Yaskawa INFORM job: DEMO_ROOF_UPPER_0625_3PAINT_53.JBI

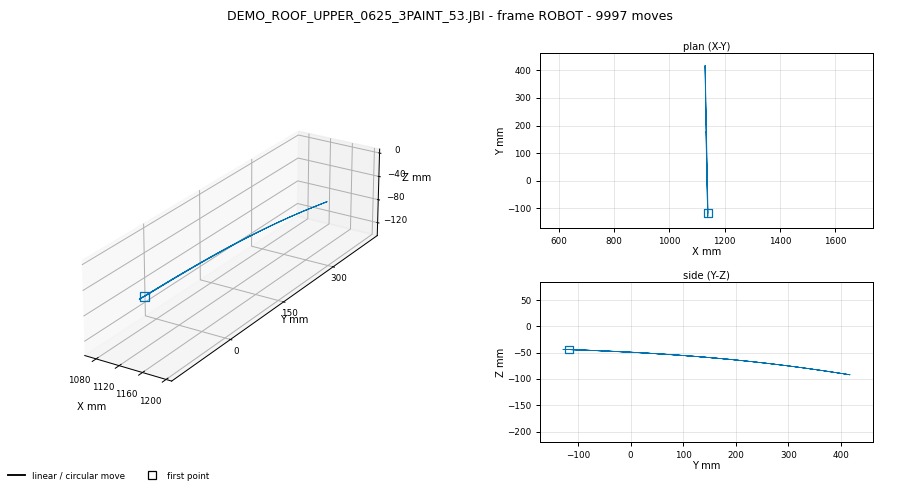
[picture p0: tool path of DEMO_ROOF_UPPER_0625_3PAINT_53.JBI in frame ROBOT, 9997 of 9997 moves have a stored position in this frame; points joined in program order, loops and branches not executed]
/JOB
//NAME DEMO_ROOF_UPPER_0625_3PAINT53
//POS
///NPOS 9997,0,0,0,0,0
///TOOL 0
///USER 0
///POSTYPE ROBOT
///RECTAN
///RCONF 1,0,0,0,0,0,0,0,0,0,0,0,0,0,0,0,0,0,0,0,0,0,0,0
C00000=1140.310,-116.948,-44.068,178.572,6.025,149.504
C00001=1140.305,-116.698,-44.077,178.574,6.025,149.503
C00002=1140.299,-116.448,-44.085,178.576,6.025,149.503
C00003=1140.294,-116.198,-44.094,178.577,6.025,149.502
C00004=1140.288,-115.949,-44.102,178.580,6.026,149.502
C00005=1140.283,-115.699,-44.111,178.581,6.026,149.501
C00006=1140.278,-115.448,-44.119,178.583,6.027,149.501
C00007=1140.272,-115.199,-44.128,178.585,6.027,149.500
C00008=1140.267,-114.949,-44.137,178.587,6.027,149.500
C00009=1140.262,-114.699,-44.146,178.589,6.028,149.499
C00010=1140.256,-114.449,-44.154,178.592,6.028,149.499
C00011=1140.250,-114.200,-44.163,178.594,6.029,149.498
C00012=1140.245,-113.950,-44.171,178.595,6.028,149.498
C00013=1140.240,-113.700,-44.180,178.598,6.029,149.497
C00014=1140.234,-113.450,-44.188,178.599,6.029,149.497
C00015=1140.229,-113.200,-44.197,178.601,6.030,149.496
C00016=1140.224,-112.951,-44.206,178.604,6.031,149.496
C00017=1140.218,-112.701,-44.215,178.605,6.031,149.495
C00018=1140.213,-112.452,-44.223,178.607,6.031,149.495
C00019=1140.208,-112.202,-44.232,178.609,6.031,149.494
C00020=1140.202,-111.951,-44.240,178.611,6.032,149.494
C00021=1140.197,-111.701,-44.249,178.613,6.032,149.493
C00022=1140.191,-111.452,-44.258,178.615,6.033,149.493
C00023=1140.186,-111.202,-44.267,178.617,6.034,149.492
C00024=1140.181,-110.953,-44.276,178.619,6.034,149.492
C00025=1140.176,-110.703,-44.285,178.621,6.034,149.491
C00026=1140.170,-110.452,-44.293,178.623,6.034,149.491
C00027=1140.164,-110.203,-44.301,178.625,6.035,149.490
C00028=1140.159,-109.953,-44.310,178.627,6.035,149.490
C00029=1140.154,-109.703,-44.319,178.629,6.035,149.489
C00030=1140.149,-109.454,-44.328,178.631,6.036,149.489
C00031=1140.143,-109.204,-44.337,178.633,6.036,149.488
C00032=1140.138,-108.955,-44.345,178.635,6.037,149.488
C00033=1140.132,-108.704,-44.355,178.637,6.037,149.487
C00034=1140.127,-108.454,-44.364,178.639,6.037,149.487
C00035=1140.122,-108.205,-44.373,178.641,6.038,149.486
C00036=1140.116,-107.955,-44.381,178.643,6.038,149.486
C00037=1140.111,-107.706,-44.390,178.645,6.039,149.485
C00038=1140.105,-107.455,-44.398,178.647,6.038,149.485
C00039=1140.100,-107.205,-44.407,178.649,6.039,149.484
C00040=1140.095,-106.955,-44.416,178.651,6.040,149.484
C00041=1140.090,-106.706,-44.425,178.653,6.040,149.483
C00042=1140.084,-106.456,-44.434,178.655,6.041,149.483
C00043=1140.078,-106.206,-44.443,178.657,6.041,149.482
C00044=1140.073,-105.956,-44.452,178.659,6.041,149.482
C00045=1140.068,-105.707,-44.461,178.661,6.042,149.481
C00046=1140.063,-105.457,-44.470,178.663,6.042,149.481
C00047=1140.057,-105.207,-44.479,178.665,6.043,149.480
C00048=1140.052,-104.958,-44.487,178.667,6.042,149.479
C00049=1140.047,-104.708,-44.496,178.669,6.043,149.479
C00050=1140.041,-104.458,-44.506,178.671,6.044,149.478
C00051=1140.035,-104.208,-44.514,178.673,6.044,149.478
C00052=1140.030,-103.958,-44.523,178.675,6.045,149.478
C00053=1140.025,-103.709,-44.533,178.677,6.045,149.477
C00054=1140.020,-103.459,-44.542,178.679,6.045,149.477
C00055=1140.014,-103.186,-44.551,178.681,6.046,149.476
C00056=1140.008,-102.915,-44.561,178.684,6.046,149.475
C00057=1140.002,-102.642,-44.571,178.685,6.046,149.475
C00058=1139.996,-102.370,-44.581,178.687,6.047,149.474
C00059=1139.991,-102.120,-44.590,178.690,6.048,149.474
C00060=1139.986,-101.870,-44.599,178.692,6.047,149.473
C00061=1139.981,-101.621,-44.608,178.694,6.048,149.473
C00062=1139.976,-101.371,-44.617,178.696,6.049,149.472
C00063=1139.970,-101.121,-44.627,178.698,6.049,149.472
C00064=1139.964,-100.872,-44.635,178.700,6.050,149.471
C00065=1139.959,-100.622,-44.644,178.702,6.050,149.471
C00066=1139.954,-100.372,-44.653,178.704,6.050,149.470
C00067=1139.948,-100.122,-44.662,178.706,6.051,149.470
C00068=1139.943,-99.872,-44.671,178.709,6.052,149.469
C00069=1139.938,-99.623,-44.681,178.710,6.051,149.469
C00070=1139.933,-99.373,-44.690,178.712,6.052,149.468
C00071=1139.927,-99.123,-44.699,178.714,6.052,149.468
C00072=1139.921,-98.873,-44.708,178.716,6.053,149.467
C00073=1139.916,-98.623,-44.717,178.718,6.054,149.467
C00074=1139.911,-98.374,-44.727,178.720,6.054,149.466
C00075=1139.906,-98.124,-44.736,178.723,6.054,149.465
C00076=1139.900,-97.874,-44.745,178.725,6.055,149.465
C00077=1139.895,-97.625,-44.754,178.726,6.055,149.464
C00078=1139.889,-97.374,-44.763,178.729,6.055,149.464
C00079=1139.884,-97.125,-44.773,178.731,6.056,149.463
C00080=1139.879,-96.875,-44.782,178.732,6.056,149.463
C00081=1139.873,-96.625,-44.791,178.735,6.057,149.463
C00082=1139.868,-96.375,-44.800,178.737,6.057,149.462
C00083=1139.862,-96.126,-44.809,178.739,6.057,149.461
C00084=1139.857,-95.876,-44.819,178.741,6.058,149.461
C00085=1139.852,-95.626,-44.828,178.743,6.058,149.460
C00086=1139.847,-95.376,-44.837,178.745,6.059,149.460
C00087=1139.841,-95.127,-44.847,178.747,6.060,149.459
C00088=1139.836,-94.877,-44.856,178.749,6.059,149.459
C00089=1139.831,-94.627,-44.865,178.751,6.060,149.458
C00090=1139.825,-94.377,-44.874,178.754,6.061,149.458
C00091=1139.820,-94.128,-44.884,178.755,6.061,149.457
C00092=1139.815,-93.878,-44.893,178.757,6.061,149.457
C00093=1139.809,-93.628,-44.902,178.760,6.062,149.456
C00094=1139.804,-93.378,-44.912,178.761,6.062,149.456
C00095=1139.799,-93.129,-44.921,178.763,6.063,149.455
C00096=1139.793,-92.878,-44.930,178.766,6.063,149.455
C00097=1139.788,-92.629,-44.940,178.768,6.063,149.454
C00098=1139.782,-92.379,-44.950,178.770,6.064,149.454
C00099=1139.777,-92.129,-44.959,178.772,6.065,149.453
C00100=1139.772,-91.880,-44.968,178.774,6.065,149.453
C00101=1139.766,-91.630,-44.978,178.776,6.065,149.452
C00102=1139.761,-91.380,-44.987,178.778,6.066,149.451
C00103=1139.755,-91.130,-44.997,178.780,6.066,149.451
C00104=1139.750,-90.880,-45.006,178.782,6.066,149.450
C00105=1139.745,-90.631,-45.015,178.784,6.067,149.450
C00106=1139.739,-90.381,-45.025,178.787,6.068,149.449
C00107=1139.734,-90.131,-45.034,178.788,6.068,149.449
C00108=1139.729,-89.882,-45.044,178.791,6.068,149.448
C00109=1139.724,-89.632,-45.053,178.793,6.069,149.448
C00110=1139.718,-89.382,-45.063,178.795,6.069,149.447
C00111=1139.713,-89.132,-45.072,178.797,6.070,149.447
C00112=1139.707,-88.883,-45.082,178.799,6.071,149.446
C00113=1139.702,-88.633,-45.091,178.801,6.070,149.446
C00114=1139.697,-88.382,-45.101,178.803,6.071,149.445
C00115=1139.692,-88.133,-45.110,178.806,6.072,149.445
C00116=1139.687,-87.883,-45.119,178.807,6.072,149.444
C00117=1139.681,-87.634,-45.130,178.809,6.072,149.444
C00118=1139.676,-87.384,-45.138,178.812,6.073,149.443
C00119=1139.670,-87.134,-45.149,178.814,6.073,149.443
C00120=1139.665,-86.884,-45.158,178.816,6.073,149.442
C00121=1139.660,-86.635,-45.168,178.818,6.074,149.442
C00122=1139.654,-86.385,-45.177,178.820,6.075,149.441
C00123=1139.649,-86.135,-45.187,178.822,6.075,149.441
C00124=1139.644,-85.886,-45.196,178.824,6.075,149.440
C00125=1139.639,-85.635,-45.206,178.827,6.076,149.439
C00126=1139.633,-85.385,-45.215,178.828,6.076,149.439
C00127=1139.628,-85.136,-45.225,178.830,6.077,149.438
C00128=1139.622,-84.886,-45.236,178.833,6.078,149.438
C00129=1139.617,-84.636,-45.245,178.835,6.078,149.437
C00130=1139.611,-84.387,-45.255,178.837,6.078,149.437
C00131=1139.606,-84.137,-45.264,178.839,6.079,149.436
C00132=1139.601,-83.888,-45.274,178.841,6.079,149.436
C00133=1139.596,-83.638,-45.283,178.843,6.079,149.435
C00134=1139.591,-83.387,-45.293,178.845,6.080,149.435
C00135=1139.586,-83.138,-45.303,178.848,6.080,149.434
C00136=1139.580,-82.888,-45.312,178.850,6.081,149.434
C00137=1139.574,-82.639,-45.323,178.851,6.081,149.433
C00138=1139.569,-82.389,-45.332,178.854,6.082,149.433
C00139=1139.563,-82.139,-45.342,178.856,6.082,149.432
C00140=1139.559,-81.890,-45.351,178.858,6.082,149.431
C00141=1139.553,-81.639,-45.361,178.860,6.083,149.431
C00142=1139.548,-81.389,-45.371,178.862,6.084,149.430
C00143=1139.543,-81.140,-45.381,178.865,6.085,149.430
C00144=1139.537,-80.890,-45.391,178.867,6.084,149.429
C00145=1139.532,-80.641,-45.400,178.869,6.085,149.429
C00146=1139.526,-80.391,-45.410,178.871,6.086,149.428
C00147=1139.521,-80.140,-45.420,178.873,6.086,149.428
C00148=1139.516,-79.891,-45.430,178.875,6.086,149.427
C00149=1139.511,-79.642,-45.440,178.877,6.087,149.427
C00150=1139.505,-79.392,-45.450,178.880,6.088,149.426
C00151=1139.500,-79.142,-45.459,178.882,6.088,149.426
C00152=1139.495,-78.892,-45.470,178.883,6.088,149.425
C00153=1139.489,-78.642,-45.480,178.886,6.089,149.425
C00154=1139.484,-78.393,-45.489,178.888,6.089,149.424
C00155=1139.479,-78.143,-45.499,178.891,6.090,149.424
C00156=1139.473,-77.894,-45.509,178.892,6.090,149.423
C00157=1139.468,-77.644,-45.518,178.894,6.091,149.423
C00158=1139.463,-77.393,-45.529,178.897,6.091,149.422
C00159=1139.456,-77.123,-45.540,178.899,6.092,149.421
C00160=1139.451,-76.851,-45.550,178.901,6.093,149.421
C00161=1139.446,-76.579,-45.561,178.904,6.093,149.420
C00162=1139.440,-76.308,-45.573,178.906,6.093,149.420
C00163=1139.434,-76.058,-45.583,178.908,6.094,149.419
C00164=1139.429,-75.808,-45.592,178.910,6.094,149.419
C00165=1139.423,-75.559,-45.602,178.913,6.095,149.418
C00166=1139.418,-75.309,-45.612,178.914,6.095,149.418
C00167=1139.413,-75.059,-45.622,178.916,6.096,149.417
C00168=1139.408,-74.810,-45.632,178.919,6.096,149.416
C00169=1139.402,-74.560,-45.642,178.921,6.097,149.416
C00170=1139.396,-74.310,-45.652,178.924,6.098,149.415
C00171=1139.391,-74.060,-45.663,178.925,6.098,149.415
C00172=1139.386,-73.811,-45.672,178.928,6.098,149.414
C00173=1139.381,-73.561,-45.682,178.930,6.099,149.414
C00174=1139.375,-73.312,-45.693,178.932,6.100,149.413
C00175=1139.370,-73.061,-45.703,178.934,6.100,149.413
C00176=1139.365,-72.812,-45.713,178.936,6.100,149.412
C00177=1139.360,-72.562,-45.722,178.939,6.101,149.412
C00178=1139.355,-72.312,-45.733,178.941,6.101,149.411
C00179=1139.349,-72.062,-45.743,178.942,6.101,149.411
C00180=1139.343,-71.813,-45.753,178.945,6.102,149.410
C00181=1139.338,-71.563,-45.763,178.947,6.103,149.409
C00182=1139.333,-71.313,-45.773,178.949,6.103,149.409
C00183=1139.328,-71.064,-45.784,178.952,6.104,149.408
C00184=1139.322,-70.814,-45.794,178.953,6.104,149.408
C00185=1139.317,-70.564,-45.804,178.956,6.104,149.407
C00186=1139.312,-70.314,-45.815,178.958,6.105,149.407
C00187=1139.307,-70.065,-45.824,178.960,6.106,149.406
C00188=1139.302,-69.815,-45.835,178.963,6.107,149.406
C00189=1139.296,-69.565,-45.845,178.965,6.106,149.405
C00190=1139.291,-69.316,-45.855,178.967,6.107,149.405
C00191=1139.285,-69.066,-45.865,178.969,6.108,149.404
C00192=1139.280,-68.816,-45.876,178.971,6.109,149.404
C00193=1139.274,-68.566,-45.886,178.974,6.109,149.403
C00194=1139.269,-68.317,-45.896,178.975,6.109,149.402
C00195=1139.265,-68.067,-45.906,178.978,6.110,149.402
C00196=1139.259,-67.817,-45.917,178.980,6.110,149.401
C00197=1139.254,-67.567,-45.927,178.982,6.111,149.401
C00198=1139.248,-67.317,-45.937,178.985,6.112,149.400
C00199=1139.243,-67.068,-45.948,178.986,6.112,149.400
C00200=1139.238,-66.818,-45.958,178.989,6.112,149.399
C00201=1139.232,-66.568,-45.968,178.991,6.113,149.399
C00202=1139.227,-66.319,-45.979,178.993,6.114,149.398
C00203=1139.222,-66.068,-45.989,178.996,6.114,149.398
C00204=1139.216,-65.819,-45.999,178.998,6.114,149.397
C00205=1139.211,-65.570,-46.009,179.000,6.115,149.396
C00206=1139.206,-65.319,-46.020,179.002,6.115,149.396
C00207=1139.201,-65.070,-46.031,179.004,6.116,149.396
C00208=1139.196,-64.820,-46.041,179.007,6.117,149.395
C00209=1139.190,-64.571,-46.051,179.008,6.117,149.394
C00210=1139.185,-64.321,-46.062,179.011,6.117,149.394
C00211=1139.180,-64.071,-46.072,179.013,6.118,149.393
C00212=1139.174,-63.821,-46.082,179.015,6.118,149.393
C00213=1139.169,-63.571,-46.093,179.018,6.119,149.392
C00214=1139.164,-63.322,-46.104,179.020,6.120,149.392
C00215=1139.158,-63.073,-46.114,179.021,6.120,149.391
C00216=1139.153,-62.822,-46.125,179.024,6.120,149.391
C00217=1139.148,-62.573,-46.135,179.026,6.121,149.390
C00218=1139.143,-62.323,-46.145,179.028,6.122,149.390
C00219=1139.137,-62.073,-46.156,179.031,6.122,149.389
C00220=1139.132,-61.823,-46.167,179.033,6.123,149.388
C00221=1139.127,-61.574,-46.177,179.035,6.123,149.388
C00222=1139.121,-61.324,-46.187,179.037,6.124,149.387
C00223=1139.116,-61.074,-46.198,179.040,6.124,149.387
C00224=1139.111,-60.825,-46.209,179.042,6.125,149.386
C00225=1139.106,-60.575,-46.219,179.044,6.126,149.386
C00226=1139.100,-60.325,-46.230,179.047,6.126,149.385
C00227=1139.095,-60.075,-46.240,179.048,6.126,149.385
C00228=1139.090,-59.826,-46.251,179.051,6.127,149.384
C00229=1139.085,-59.576,-46.262,179.053,6.128,149.384
C00230=1139.079,-59.326,-46.272,179.055,6.128,149.383
C00231=1139.074,-59.076,-46.282,179.058,6.129,149.382
C00232=1139.068,-58.827,-46.294,179.060,6.130,149.382
C00233=1139.063,-58.577,-46.305,179.062,6.130,149.381
C00234=1139.058,-58.327,-46.315,179.064,6.130,149.381
C00235=1139.053,-58.077,-46.326,179.066,6.131,149.380
C00236=1139.047,-57.828,-46.336,179.069,6.131,149.380
C00237=1139.042,-57.578,-46.347,179.071,6.132,149.379
C00238=1139.037,-57.329,-46.358,179.073,6.133,149.379
C00239=1139.032,-57.079,-46.368,179.076,6.133,149.378
C00240=1139.026,-56.829,-46.379,179.078,6.134,149.377
C00241=1139.022,-56.579,-46.390,179.080,6.134,149.377
C00242=1139.016,-56.330,-46.400,179.082,6.135,149.376
C00243=1139.011,-56.080,-46.412,179.084,6.135,149.376
C00244=1139.005,-55.830,-46.422,179.087,6.136,149.375
C00245=1139.000,-55.580,-46.433,179.089,6.136,149.375
C00246=1138.995,-55.331,-46.444,179.091,6.137,149.374
C00247=1138.990,-55.081,-46.454,179.094,6.138,149.374
C00248=1138.985,-54.832,-46.465,179.096,6.138,149.373
C00249=1138.980,-54.582,-46.476,179.098,6.138,149.373
C00250=1138.973,-54.332,-46.486,179.100,6.139,149.372
C00251=1138.969,-54.082,-46.498,179.103,6.140,149.371
C00252=1138.964,-53.832,-46.508,179.105,6.140,149.371
C00253=1138.958,-53.583,-46.519,179.107,6.141,149.371
C00254=1138.953,-53.333,-46.530,179.110,6.141,149.370
C00255=1138.947,-53.084,-46.541,179.112,6.142,149.369
C00256=1138.942,-52.833,-46.552,179.114,6.143,149.369
C00257=1138.937,-52.584,-46.563,179.116,6.143,149.368
C00258=1138.932,-52.334,-46.573,179.118,6.143,149.368
C00259=1138.927,-52.085,-46.584,179.120,6.144,149.367
C00260=1138.921,-51.835,-46.596,179.123,6.145,149.367
C00261=1138.916,-51.585,-46.607,179.125,6.145,149.366
C00262=1138.911,-51.336,-46.617,179.127,6.146,149.366
C00263=1138.905,-51.065,-46.629,179.130,6.146,149.365
C00264=1138.899,-50.794,-46.641,179.132,6.147,149.364
C00265=1138.894,-50.524,-46.653,179.135,6.148,149.364
C00266=1138.888,-50.253,-46.665,179.137,6.148,149.363
C00267=1138.883,-50.003,-46.675,179.139,6.149,149.363
C00268=1138.877,-49.753,-46.687,179.142,6.150,149.362
C00269=1138.872,-49.503,-46.698,179.144,6.150,149.362
C00270=1138.867,-49.254,-46.709,179.146,6.151,149.361
C00271=1138.861,-49.003,-46.720,179.149,6.151,149.360
C00272=1138.856,-48.755,-46.731,179.151,6.152,149.360
C00273=1138.851,-48.505,-46.742,179.153,6.152,149.359
C00274=1138.846,-48.255,-46.753,179.155,6.153,149.359
C00275=1138.840,-48.005,-46.764,179.158,6.153,149.358
C00276=1138.836,-47.756,-46.775,179.160,6.154,149.358
C00277=1138.831,-47.506,-46.786,179.162,6.155,149.357
C00278=1138.825,-47.256,-46.798,179.165,6.155,149.357
C00279=1138.820,-47.006,-46.808,179.167,6.156,149.356
C00280=1138.814,-46.757,-46.819,179.169,6.157,149.356
C00281=1138.809,-46.507,-46.831,179.172,6.157,149.355
C00282=1138.804,-46.257,-46.841,179.174,6.158,149.354
C00283=1138.799,-46.008,-46.852,179.176,6.159,149.354
C00284=1138.793,-45.758,-46.864,179.179,6.159,149.353
C00285=1138.788,-45.508,-46.876,179.181,6.160,149.353
C00286=1138.782,-45.259,-46.886,179.183,6.160,149.352
C00287=1138.777,-45.009,-46.898,179.185,6.160,149.352
C00288=1138.773,-44.759,-46.909,179.188,6.161,149.351
C00289=1138.767,-44.509,-46.920,179.190,6.162,149.351
C00290=1138.762,-44.260,-46.931,179.192,6.162,149.350
C00291=1138.757,-44.010,-46.942,179.195,6.163,149.349
C00292=1138.752,-43.760,-46.954,179.197,6.164,149.349
C00293=1138.746,-43.511,-46.964,179.199,6.164,149.348
C00294=1138.740,-43.261,-46.976,179.202,6.165,149.348
C00295=1138.736,-43.011,-46.988,179.204,6.166,149.347
C00296=1138.731,-42.762,-46.999,179.206,6.167,149.347
C00297=1138.725,-42.512,-47.010,179.209,6.167,149.346
C00298=1138.720,-42.262,-47.021,179.211,6.168,149.346
C00299=1138.715,-42.012,-47.033,179.213,6.169,149.345
C00300=1138.709,-41.763,-47.044,179.216,6.169,149.344
C00301=1138.704,-41.513,-47.056,179.218,6.170,149.344
C00302=1138.699,-41.264,-47.067,179.220,6.171,149.344
C00303=1138.694,-41.013,-47.078,179.223,6.171,149.343
C00304=1138.688,-40.764,-47.089,179.224,6.171,149.342
C00305=1138.683,-40.514,-47.101,179.226,6.172,149.342
C00306=1138.678,-40.265,-47.112,179.229,6.172,149.341
C00307=1138.672,-40.015,-47.124,179.231,6.173,149.341
C00308=1138.667,-39.766,-47.135,179.234,6.174,149.340
C00309=1138.662,-39.516,-47.147,179.236,6.174,149.340
C00310=1138.657,-39.266,-47.158,179.238,6.175,149.339
C00311=1138.651,-39.016,-47.169,179.241,6.176,149.339
C00312=1138.646,-38.767,-47.180,179.243,6.176,149.338
C00313=1138.641,-38.517,-47.192,179.245,6.177,149.337
C00314=1138.636,-38.267,-47.204,179.248,6.178,149.337
C00315=1138.631,-38.017,-47.215,179.250,6.178,149.336
C00316=1138.625,-37.768,-47.226,179.252,6.179,149.336
C00317=1138.620,-37.518,-47.238,179.255,6.180,149.335
C00318=1138.615,-37.269,-47.249,179.257,6.180,149.335
C00319=1138.610,-37.019,-47.261,179.260,6.181,149.334
C00320=1138.605,-36.769,-47.273,179.262,6.182,149.334
C00321=1138.599,-36.520,-47.284,179.264,6.182,149.333
C00322=1138.594,-36.270,-47.296,179.267,6.183,149.332
C00323=1138.589,-36.020,-47.307,179.269,6.183,149.332
C00324=1138.584,-35.770,-47.319,179.271,6.184,149.331
C00325=1138.579,-35.521,-47.331,179.274,6.185,149.331
C00326=1138.573,-35.272,-47.342,179.276,6.185,149.330
C00327=1138.567,-35.022,-47.354,179.278,6.186,149.330
C00328=1138.563,-34.772,-47.365,179.281,6.187,149.329
C00329=1138.557,-34.522,-47.377,179.283,6.187,149.329
C00330=1138.553,-34.272,-47.388,179.285,6.188,149.328
C00331=1138.547,-34.023,-47.400,179.288,6.189,149.327
C00332=1138.541,-33.773,-47.412,179.290,6.189,149.327
C00333=1138.536,-33.524,-47.423,179.293,6.190,149.326
C00334=1138.531,-33.274,-47.435,179.295,6.191,149.326
C00335=1138.526,-33.024,-47.447,179.297,6.191,149.325
C00336=1138.521,-32.774,-47.458,179.300,6.192,149.325
C00337=1138.515,-32.524,-47.470,179.302,6.193,149.324
C00338=1138.511,-32.275,-47.481,179.304,6.193,149.324
C00339=1138.505,-32.026,-47.494,179.307,6.194,149.323
C00340=1138.500,-31.776,-47.505,179.309,6.195,149.323
C00341=1138.495,-31.526,-47.517,179.311,6.195,149.322
C00342=1138.489,-31.277,-47.529,179.314,6.196,149.321
C00343=1138.484,-31.027,-47.541,179.316,6.196,149.321
C00344=1138.479,-30.777,-47.552,179.318,6.197,149.320
C00345=1138.474,-30.527,-47.564,179.321,6.198,149.320
C00346=1138.469,-30.278,-47.576,179.323,6.198,149.319
C00347=1138.463,-30.028,-47.588,179.325,6.199,149.319
C00348=1138.458,-29.779,-47.599,179.328,6.200,149.318
C00349=1138.453,-29.529,-47.611,179.330,6.200,149.318
C00350=1138.447,-29.279,-47.623,179.333,6.201,149.317
C00351=1138.442,-29.030,-47.635,179.335,6.202,149.316
C00352=1138.437,-28.780,-47.647,179.337,6.202,149.316
C00353=1138.432,-28.530,-47.659,179.340,6.203,149.315
C00354=1138.427,-28.280,-47.671,179.342,6.204,149.315
C00355=1138.422,-28.031,-47.683,179.344,6.204,149.314
C00356=1138.417,-27.781,-47.694,179.347,6.205,149.314
C00357=1138.411,-27.531,-47.706,179.349,6.206,149.313
C00358=1138.406,-27.281,-47.718,179.351,6.206,149.313
C00359=1138.401,-27.032,-47.731,179.354,6.207,149.312
C00360=1138.396,-26.782,-47.742,179.356,6.208,149.311
C00361=1138.391,-26.532,-47.754,179.359,6.209,149.311
C00362=1138.386,-26.283,-47.767,179.361,6.210,149.310
C00363=1138.380,-26.033,-47.778,179.363,6.210,149.310
C00364=1138.375,-25.784,-47.790,179.366,6.211,149.309
C00365=1138.370,-25.534,-47.802,179.368,6.212,149.309
C00366=1138.365,-25.284,-47.814,179.370,6.212,149.308
C00367=1138.359,-25.015,-47.827,179.373,6.213,149.307
C00368=1138.354,-24.744,-47.840,179.375,6.214,149.307
C00369=1138.347,-24.474,-47.853,179.378,6.214,149.306
C00370=1138.342,-24.204,-47.866,179.381,6.216,149.306
C00371=1138.337,-23.955,-47.879,179.383,6.216,149.305
C00372=1138.331,-23.705,-47.890,179.386,6.217,149.305
C00373=1138.326,-23.455,-47.902,179.388,6.217,149.304
C00374=1138.321,-23.206,-47.914,179.390,6.218,149.304
C00375=1138.316,-22.956,-47.926,179.393,6.219,149.303
C00376=1138.311,-22.707,-47.939,179.395,6.219,149.303
C00377=1138.305,-22.457,-47.951,179.397,6.220,149.302
C00378=1138.300,-22.207,-47.963,179.400,6.221,149.301
C00379=1138.295,-21.957,-47.975,179.402,6.221,149.301
C00380=1138.289,-21.707,-47.987,179.405,6.222,149.300
C00381=1138.284,-21.458,-48.000,179.407,6.223,149.300
C00382=1138.280,-21.208,-48.011,179.409,6.223,149.299
C00383=1138.274,-20.959,-48.024,179.412,6.225,149.299
C00384=1138.269,-20.709,-48.035,179.414,6.225,149.298
C00385=1138.264,-20.460,-48.048,179.417,6.226,149.297
C00386=1138.258,-20.210,-48.060,179.419,6.227,149.297
C00387=1138.253,-19.961,-48.073,179.421,6.227,149.296
C00388=1138.248,-19.710,-48.085,179.424,6.228,149.296
C00389=1138.243,-19.461,-48.097,179.426,6.229,149.295
C00390=1138.238,-19.211,-48.109,179.428,6.229,149.295
C00391=1138.233,-18.961,-48.122,179.431,6.230,149.294
C00392=1138.228,-18.712,-48.134,179.433,6.231,149.294
C00393=1138.222,-18.462,-48.146,179.436,6.231,149.293
C00394=1138.217,-18.213,-48.159,179.439,6.233,149.293
C00395=1138.212,-17.963,-48.171,179.441,6.233,149.292
C00396=1138.207,-17.714,-48.183,179.444,6.234,149.291
C00397=1138.201,-17.464,-48.195,179.446,6.235,149.291
C00398=1138.196,-17.214,-48.208,179.448,6.235,149.290
C00399=1138.191,-16.965,-48.221,179.451,6.236,149.290
C00400=1138.186,-16.714,-48.233,179.453,6.237,149.289
C00401=1138.181,-16.465,-48.245,179.455,6.237,149.289
C00402=1138.175,-16.215,-48.257,179.458,6.238,149.288
C00403=1138.170,-15.966,-48.270,179.460,6.239,149.288
C00404=1138.165,-15.717,-48.282,179.463,6.240,149.287
C00405=1138.160,-15.467,-48.294,179.465,6.241,149.286
C00406=1138.155,-15.217,-48.307,179.467,6.241,149.286
C00407=1138.150,-14.967,-48.320,179.470,6.242,149.285
C00408=1138.145,-14.717,-48.332,179.472,6.243,149.285
C00409=1138.140,-14.468,-48.344,179.474,6.243,149.284
C00410=1138.134,-14.219,-48.357,179.477,6.244,149.284
C00411=1138.129,-13.969,-48.370,179.479,6.245,149.283
C00412=1138.123,-13.719,-48.382,179.481,6.245,149.283
C00413=1138.118,-13.470,-48.395,179.485,6.247,149.282
C00414=1138.114,-13.220,-48.408,179.487,6.247,149.282
C00415=1138.108,-12.970,-48.420,179.490,6.248,149.281
C00416=1138.103,-12.721,-48.432,179.492,6.249,149.280
C00417=1138.098,-12.471,-48.445,179.494,6.249,149.280
C00418=1138.093,-12.222,-48.457,179.497,6.250,149.279
C00419=1138.088,-11.972,-48.470,179.499,6.251,149.279
C00420=1138.082,-11.722,-48.483,179.501,6.252,149.278
C00421=1138.077,-11.472,-48.495,179.504,6.253,149.278
C00422=1138.072,-11.223,-48.508,179.506,6.253,149.277
C00423=1138.067,-10.974,-48.521,179.509,6.254,149.277
C00424=1138.062,-10.724,-48.534,179.511,6.255,149.276
C00425=1138.057,-10.474,-48.545,179.513,6.255,149.275
C00426=1138.052,-10.224,-48.558,179.516,6.256,149.275
C00427=1138.046,-9.975,-48.571,179.519,6.257,149.274
C00428=1138.041,-9.725,-48.584,179.521,6.258,149.274
C00429=1138.036,-9.475,-48.597,179.524,6.259,149.273
C00430=1138.031,-9.226,-48.609,179.526,6.260,149.273
C00431=1138.026,-8.976,-48.621,179.528,6.260,149.272
C00432=1138.020,-8.727,-48.634,179.531,6.261,149.272
C00433=1138.015,-8.477,-48.647,179.533,6.262,149.271
C00434=1138.010,-8.227,-48.660,179.536,6.263,149.271
C00435=1138.005,-7.978,-48.673,179.538,6.264,149.270
C00436=1138.000,-7.729,-48.685,179.540,6.264,149.269
C00437=1137.995,-7.478,-48.699,179.543,6.265,149.269
C00438=1137.989,-7.229,-48.711,179.545,6.266,149.268
C00439=1137.984,-6.980,-48.724,179.547,6.266,149.268
C00440=1137.979,-6.730,-48.737,179.551,6.268,149.267
C00441=1137.974,-6.480,-48.750,179.553,6.268,149.267
C00442=1137.969,-6.231,-48.763,179.555,6.269,149.266
C00443=1137.964,-5.981,-48.775,179.558,6.270,149.266
C00444=1137.959,-5.731,-48.788,179.560,6.270,149.265
C00445=1137.953,-5.482,-48.802,179.563,6.272,149.265
C00446=1137.948,-5.232,-48.814,179.565,6.272,149.264
C00447=1137.943,-4.983,-48.827,179.568,6.273,149.263
C00448=1137.938,-4.733,-48.840,179.570,6.274,149.263
C00449=1137.933,-4.483,-48.853,179.572,6.274,149.262
C00450=1137.928,-4.234,-48.866,179.575,6.275,149.262
C00451=1137.922,-3.984,-48.879,179.578,6.276,149.261
C00452=1137.917,-3.734,-48.892,179.580,6.277,149.261
C00453=1137.912,-3.485,-48.904,179.582,6.278,149.260
C00454=1137.907,-3.235,-48.918,179.585,6.278,149.259
C00455=1137.902,-2.985,-48.930,179.587,6.279,149.259
C00456=1137.896,-2.736,-48.943,179.590,6.280,149.258
C00457=1137.891,-2.486,-48.957,179.592,6.281,149.258
C00458=1137.886,-2.236,-48.969,179.595,6.282,149.257
C00459=1137.881,-1.987,-48.982,179.597,6.283,149.257
C00460=1137.876,-1.737,-48.996,179.599,6.283,149.256
C00461=1137.871,-1.488,-49.009,179.602,6.285,149.256
C00462=1137.865,-1.239,-49.022,179.605,6.285,149.255
C00463=1137.861,-0.989,-49.035,179.607,6.286,149.255
C00464=1137.855,-0.739,-49.047,179.609,6.287,149.254
C00465=1137.850,-0.489,-49.061,179.612,6.287,149.253
C00466=1137.845,-0.240,-49.074,179.615,6.289,149.253
C00467=1137.839,0.009,-49.088,179.617,6.289,149.252
C00468=1137.835,0.259,-49.100,179.619,6.290,149.252
C00469=1137.829,0.509,-49.114,179.622,6.291,149.251
C00470=1137.824,0.758,-49.126,179.624,6.291,149.251
C00471=1137.819,1.028,-49.141,179.627,6.293,149.250
C00472=1137.814,1.298,-49.155,179.630,6.293,149.250
C00473=1137.808,1.568,-49.169,179.633,6.295,149.249
C00474=1137.802,1.836,-49.184,179.635,6.295,149.248
C00475=1137.797,2.086,-49.197,179.637,6.296,149.248
C00476=1137.791,2.336,-49.210,179.641,6.297,149.247
C00477=1137.787,2.585,-49.224,179.643,6.298,149.247
C00478=1137.781,2.835,-49.237,179.645,6.299,149.246
C00479=1137.776,3.084,-49.249,179.648,6.300,149.246
C00480=1137.772,3.334,-49.262,179.650,6.300,149.245
C00481=1137.766,3.583,-49.276,179.653,6.302,149.245
C00482=1137.761,3.834,-49.290,179.655,6.302,149.244
C00483=1137.756,4.083,-49.303,179.657,6.303,149.244
C00484=1137.751,4.333,-49.317,179.660,6.304,149.243
C00485=1137.746,4.582,-49.329,179.663,6.305,149.242
C00486=1137.740,4.832,-49.343,179.665,6.306,149.242
C00487=1137.736,5.081,-49.356,179.668,6.306,149.241
C00488=1137.730,5.331,-49.370,179.670,6.307,149.241
C00489=1137.725,5.580,-49.383,179.673,6.309,149.240
C00490=1137.720,5.830,-49.396,179.675,6.309,149.240
C00491=1137.715,6.080,-49.409,179.677,6.310,149.239
C00492=1137.710,6.329,-49.423,179.680,6.311,149.239
C00493=1137.704,6.579,-49.437,179.683,6.312,149.238
C00494=1137.699,6.828,-49.450,179.685,6.313,149.238
C00495=1137.694,7.078,-49.464,179.688,6.313,149.237
C00496=1137.689,7.327,-49.476,179.690,6.314,149.236
C00497=1137.684,7.577,-49.491,179.693,6.316,149.236
C00498=1137.678,7.827,-49.504,179.695,6.316,149.235
C00499=1137.674,8.076,-49.517,179.697,6.317,149.235
C00500=1137.668,8.326,-49.531,179.700,6.319,149.234
C00501=1137.664,8.575,-49.544,179.703,6.319,149.234
C00502=1137.659,8.826,-49.558,179.705,6.320,149.233
C00503=1137.653,9.075,-49.572,179.708,6.320,149.232
C00504=1137.649,9.325,-49.585,179.711,6.322,149.232
C00505=1137.643,9.574,-49.599,179.713,6.323,149.232
C00506=1137.638,9.824,-49.612,179.715,6.323,149.231
C00507=1137.633,10.073,-49.626,179.718,6.324,149.230
C00508=1137.628,10.323,-49.639,179.720,6.326,149.230
C00509=1137.622,10.572,-49.653,179.723,6.326,149.229
C00510=1137.618,10.821,-49.667,179.725,6.327,149.229
C00511=1137.612,11.071,-49.680,179.728,6.328,149.228
C00512=1137.607,11.321,-49.694,179.731,6.329,149.228
C00513=1137.603,11.571,-49.707,179.733,6.330,149.227
C00514=1137.597,11.820,-49.721,179.735,6.330,149.226
C00515=1137.592,12.070,-49.735,179.738,6.332,149.226
C00516=1137.586,12.319,-49.749,179.740,6.332,149.226
C00517=1137.582,12.568,-49.762,179.743,6.333,149.225
C00518=1137.577,12.819,-49.776,179.746,6.335,149.224
C00519=1137.571,13.068,-49.790,179.748,6.335,149.224
C00520=1137.566,13.317,-49.804,179.751,6.336,149.223
C00521=1137.561,13.567,-49.817,179.753,6.337,149.223
C00522=1137.556,13.816,-49.831,179.756,6.338,149.222
C00523=1137.551,14.066,-49.845,179.758,6.339,149.222
C00524=1137.545,14.316,-49.858,179.760,6.339,149.221
C00525=1137.541,14.565,-49.872,179.764,6.341,149.221
C00526=1137.536,14.814,-49.886,179.766,6.341,149.220
C00527=1137.530,15.065,-49.899,179.768,6.342,149.220
C00528=1137.525,15.314,-49.914,179.771,6.344,149.219
C00529=1137.520,15.563,-49.928,179.773,6.344,149.218
C00530=1137.516,15.813,-49.941,179.776,6.345,149.218
C00531=1137.510,16.063,-49.955,179.779,6.346,149.217
C00532=1137.505,16.312,-49.969,179.781,6.347,149.217
C00533=1137.500,16.562,-49.983,179.783,6.348,149.216
C00534=1137.495,16.811,-49.997,179.786,6.349,149.216
C00535=1137.489,17.060,-50.011,179.789,6.350,149.215
C00536=1137.485,17.310,-50.024,179.791,6.351,149.215
C00537=1137.480,17.560,-50.039,179.794,6.352,149.214
C00538=1137.474,17.809,-50.052,179.796,6.353,149.214
C00539=1137.469,18.059,-50.067,179.799,6.353,149.213
C00540=1137.464,18.309,-50.081,179.802,6.355,149.213
C00541=1137.458,18.558,-50.094,179.804,6.356,149.212
C00542=1137.454,18.808,-50.108,179.806,6.356,149.211
C00543=1137.449,19.058,-50.123,179.809,6.358,149.211
C00544=1137.444,19.306,-50.136,179.811,6.359,149.210
C00545=1137.439,19.556,-50.150,179.814,6.359,149.210
C00546=1137.434,19.806,-50.165,179.817,6.361,149.209
C00547=1137.429,20.056,-50.179,179.819,6.362,149.209
C00548=1137.423,20.305,-50.193,179.822,6.362,149.208
C00549=1137.418,20.555,-50.206,179.824,6.364,149.208
C00550=1137.413,20.805,-50.221,179.827,6.364,149.207
C00551=1137.408,21.054,-50.235,179.829,6.365,149.207
C00552=1137.403,21.303,-50.249,179.832,6.366,149.206
C00553=1137.398,21.553,-50.263,179.835,6.367,149.205
C00554=1137.393,21.803,-50.277,179.837,6.369,149.205
C00555=1137.388,22.052,-50.292,179.840,6.369,149.205
C00556=1137.382,22.301,-50.306,179.842,6.370,149.204
C00557=1137.377,22.551,-50.320,179.845,6.371,149.203
C00558=1137.372,22.801,-50.334,179.847,6.372,149.203
C00559=1137.367,23.051,-50.348,179.850,6.373,149.202
C00560=1137.362,23.300,-50.362,179.853,6.374,149.202
C00561=1137.357,23.549,-50.377,179.855,6.375,149.201
C00562=1137.352,23.799,-50.391,179.858,6.376,149.201
C00563=1137.347,24.049,-50.405,179.860,6.377,149.200
C00564=1137.341,24.298,-50.419,179.862,6.378,149.200
C00565=1137.336,24.547,-50.433,179.866,6.379,149.199
C00566=1137.331,24.797,-50.448,179.868,6.380,149.199
C00567=1137.327,25.046,-50.463,179.870,6.380,149.198
C00568=1137.322,25.296,-50.477,179.873,6.382,149.197
C00569=1137.316,25.545,-50.491,179.875,6.383,149.197
C00570=1137.311,25.795,-50.505,179.879,6.384,149.196
C00571=1137.306,26.044,-50.519,179.881,6.385,149.196
C00572=1137.301,26.294,-50.534,179.883,6.386,149.195
C00573=1137.296,26.544,-50.548,179.886,6.387,149.195
C00574=1137.292,26.793,-50.562,179.888,6.388,149.194
C00575=1137.285,27.062,-50.578,179.892,6.389,149.194
C00576=1137.280,27.331,-50.594,179.894,6.390,149.193
C00577=1137.274,27.600,-50.609,179.897,6.391,149.192
C00578=1137.269,27.869,-50.625,179.900,6.393,149.192
C00579=1137.264,28.119,-50.639,179.902,6.394,149.192
C00580=1137.259,28.369,-50.654,179.905,6.394,149.191
C00581=1137.254,28.618,-50.668,179.907,6.396,149.190
C00582=1137.249,28.867,-50.683,179.910,6.396,149.190
C00583=1137.244,29.116,-50.697,179.913,6.398,149.189
C00584=1137.239,29.366,-50.711,179.915,6.399,149.189
C00585=1137.234,29.616,-50.725,179.918,6.399,149.188
C00586=1137.228,29.865,-50.741,179.920,6.401,149.188
C00587=1137.223,30.115,-50.755,179.922,6.401,149.187
C00588=1137.218,30.365,-50.770,179.926,6.403,149.187
C00589=1137.213,30.614,-50.784,179.928,6.403,149.186
C00590=1137.209,30.863,-50.799,179.930,6.404,149.186
C00591=1137.203,31.113,-50.814,179.933,6.406,149.185
C00592=1137.197,31.363,-50.828,179.935,6.406,149.185
C00593=1137.193,31.612,-50.843,179.938,6.408,149.184
C00594=1137.188,31.861,-50.857,179.941,6.408,149.183
C00595=1137.183,32.111,-50.871,179.944,6.410,149.183
C00596=1137.178,32.360,-50.887,179.946,6.411,149.183
C00597=1137.173,32.610,-50.901,179.949,6.412,149.182
C00598=1137.168,32.860,-50.915,179.951,6.413,149.181
C00599=1137.163,33.109,-50.930,179.953,6.414,149.181
C00600=1137.157,33.359,-50.945,179.957,6.415,149.180
C00601=1137.153,33.608,-50.960,179.959,6.416,149.180
C00602=1137.148,33.858,-50.974,179.962,6.417,149.179
C00603=1137.142,34.108,-50.989,179.964,6.418,149.179
C00604=1137.137,34.357,-51.004,179.967,6.420,149.178
C00605=1137.132,34.607,-51.019,179.969,6.420,149.178
C00606=1137.128,34.856,-51.034,179.972,6.422,149.177
C00607=1137.122,35.106,-51.048,179.975,6.422,149.177
C00608=1137.117,35.355,-51.063,179.977,6.423,149.176
C00609=1137.112,35.604,-51.078,179.980,6.425,149.176
C00610=1137.107,35.854,-51.093,179.982,6.425,149.175
C00611=1137.102,36.104,-51.108,179.985,6.427,149.175
C00612=1137.097,36.353,-51.123,179.988,6.427,149.174
C00613=1137.092,36.603,-51.137,179.990,6.429,149.174
C00614=1137.087,36.852,-51.152,179.992,6.430,149.173
C00615=1137.081,37.102,-51.167,179.996,6.431,149.172
C00616=1137.077,37.351,-51.182,179.998,6.432,149.172
C00617=1137.072,37.601,-51.197,-179.999,6.434,149.171
C00618=1137.066,37.850,-51.212,-179.997,6.434,149.171
C00619=1137.061,38.100,-51.226,-179.994,6.436,149.170
C00620=1137.057,38.349,-51.241,-179.992,6.437,149.170
C00621=1137.051,38.598,-51.257,-179.989,6.438,149.169
C00622=1137.046,38.848,-51.271,-179.986,6.439,149.169
C00623=1137.041,39.097,-51.287,-179.984,6.439,149.168
C00624=1137.036,39.347,-51.301,-179.981,6.441,149.168
C00625=1137.031,39.596,-51.317,-179.979,6.441,149.167
C00626=1137.026,39.846,-51.332,-179.976,6.443,149.167
C00627=1137.021,40.095,-51.346,-179.973,6.444,149.166
C00628=1137.016,40.345,-51.362,-179.971,6.445,149.166
C00629=1137.011,40.594,-51.377,-179.968,6.446,149.165
C00630=1137.005,40.844,-51.391,-179.965,6.447,149.165
C00631=1137.001,41.093,-51.406,-179.963,6.448,149.164
C00632=1136.995,41.342,-51.422,-179.960,6.450,149.164
C00633=1136.991,41.593,-51.437,-179.958,6.450,149.163
C00634=1136.986,41.842,-51.452,-179.955,6.452,149.163
C00635=1136.981,42.091,-51.467,-179.953,6.453,149.162
C00636=1136.975,42.341,-51.482,-179.949,6.454,149.161
C00637=1136.971,42.590,-51.497,-179.947,6.455,149.161
C00638=1136.965,42.840,-51.513,-179.945,6.456,149.160
C00639=1136.961,43.089,-51.528,-179.942,6.457,149.160
C00640=1136.955,43.339,-51.543,-179.939,6.458,149.159
C00641=1136.950,43.588,-51.558,-179.937,6.459,149.159
C00642=1136.946,43.838,-51.574,-179.934,6.461,149.158
C00643=1136.940,44.087,-51.589,-179.932,6.461,149.158
C00644=1136.935,44.336,-51.604,-179.929,6.463,149.157
C00645=1136.930,44.587,-51.619,-179.926,6.464,149.157
C00646=1136.925,44.836,-51.634,-179.923,6.465,149.156
C00647=1136.920,45.085,-51.650,-179.921,6.467,149.156
C00648=1136.916,45.335,-51.665,-179.918,6.467,149.155
C00649=1136.910,45.584,-51.680,-179.915,6.469,149.155
C00650=1136.905,45.834,-51.696,-179.913,6.470,149.154
C00651=1136.900,46.083,-51.711,-179.910,6.471,149.154
C00652=1136.895,46.333,-51.726,-179.908,6.472,149.153
C00653=1136.890,46.582,-51.741,-179.905,6.473,149.153
C00654=1136.885,46.832,-51.757,-179.903,6.474,149.152
C00655=1136.880,47.081,-51.772,-179.900,6.475,149.152
C00656=1136.875,47.330,-51.787,-179.897,6.476,149.151
C00657=1136.870,47.580,-51.803,-179.895,6.478,149.151
C00658=1136.864,47.829,-51.819,-179.892,6.478,149.150
C00659=1136.860,48.079,-51.834,-179.889,6.480,149.150
C00660=1136.855,48.328,-51.850,-179.886,6.482,149.149
C00661=1136.850,48.578,-51.865,-179.884,6.482,149.148
C00662=1136.845,48.827,-51.880,-179.881,6.484,149.148
C00663=1136.840,49.077,-51.896,-179.879,6.485,149.148
C00664=1136.835,49.326,-51.912,-179.876,6.486,149.147
C00665=1136.830,49.575,-51.927,-179.874,6.487,149.146
C00666=1136.825,49.825,-51.942,-179.871,6.488,149.146
C00667=1136.819,50.074,-51.958,-179.869,6.489,149.146
C00668=1136.815,50.324,-51.973,-179.865,6.490,149.145
C00669=1136.810,50.573,-51.989,-179.863,6.492,149.144
C00670=1136.804,50.823,-52.004,-179.860,6.493,149.144
C00671=1136.800,51.073,-52.020,-179.857,6.494,149.143
C00672=1136.795,51.322,-52.035,-179.855,6.495,149.143
C00673=1136.790,51.571,-52.051,-179.852,6.497,149.142
C00674=1136.784,51.821,-52.067,-179.850,6.497,149.142
C00675=1136.779,52.071,-52.083,-179.847,6.499,149.141
C00676=1136.775,52.319,-52.098,-179.844,6.500,149.141
C00677=1136.770,52.569,-52.114,-179.841,6.501,149.140
C00678=1136.764,52.818,-52.129,-179.839,6.502,149.140
C00679=1136.759,53.087,-52.147,-179.836,6.504,149.139
C00680=1136.754,53.356,-52.164,-179.833,6.505,149.139
C00681=1136.748,53.625,-52.180,-179.831,6.506,149.138
C00682=1136.743,53.893,-52.197,-179.827,6.507,149.138
C00683=1136.738,54.142,-52.213,-179.825,6.509,149.137
C00684=1136.733,54.392,-52.229,-179.822,6.510,149.137
C00685=1136.728,54.641,-52.244,-179.819,6.511,149.136
C00686=1136.722,54.891,-52.260,-179.817,6.512,149.136
C00687=1136.718,55.141,-52.276,-179.814,6.514,149.135
C00688=1136.713,55.389,-52.292,-179.812,6.515,149.135
C00689=1136.708,55.639,-52.307,-179.809,6.516,149.134
C00690=1136.703,55.889,-52.323,-179.806,6.517,149.134
C00691=1136.698,56.138,-52.339,-179.804,6.518,149.133
C00692=1136.693,56.387,-52.355,-179.801,6.520,149.132
C00693=1136.688,56.637,-52.371,-179.798,6.521,149.132
C00694=1136.683,56.887,-52.387,-179.796,6.522,149.132
C00695=1136.678,57.136,-52.403,-179.793,6.523,149.131
C00696=1136.673,57.386,-52.419,-179.790,6.524,149.130
C00697=1136.667,57.635,-52.434,-179.788,6.526,149.130
C00698=1136.664,57.884,-52.450,-179.785,6.527,149.130
C00699=1136.658,58.134,-52.466,-179.782,6.528,149.129
C00700=1136.653,58.384,-52.482,-179.780,6.529,149.128
C00701=1136.648,58.632,-52.498,-179.777,6.530,149.128
C00702=1136.643,58.882,-52.514,-179.775,6.532,149.128
C00703=1136.638,59.132,-52.530,-179.771,6.533,149.127
C00704=1136.633,59.381,-52.546,-179.769,6.534,149.126
C00705=1136.628,59.631,-52.562,-179.766,6.536,149.126
C00706=1136.623,59.880,-52.578,-179.763,6.537,149.125
C00707=1136.618,60.129,-52.594,-179.761,6.538,149.125
C00708=1136.613,60.379,-52.610,-179.758,6.539,149.125
C00709=1136.608,60.628,-52.626,-179.756,6.541,149.124
C00710=1136.603,60.878,-52.642,-179.753,6.542,149.123
C00711=1136.598,61.127,-52.659,-179.750,6.543,149.123
C00712=1136.593,61.377,-52.675,-179.748,6.544,149.123
C00713=1136.588,61.626,-52.691,-179.745,6.545,149.122
C00714=1136.583,61.876,-52.707,-179.742,6.547,149.121
C00715=1136.578,62.125,-52.723,-179.740,6.548,149.121
C00716=1136.573,62.374,-52.739,-179.737,6.549,149.121
C00717=1136.568,62.623,-52.755,-179.734,6.551,149.120
C00718=1136.563,62.873,-52.771,-179.732,6.552,149.119
C00719=1136.559,63.122,-52.788,-179.729,6.553,149.119
C00720=1136.552,63.372,-52.804,-179.726,6.555,149.119
C00721=1136.548,63.622,-52.820,-179.724,6.555,149.118
C00722=1136.543,63.870,-52.837,-179.721,6.557,149.117
C00723=1136.538,64.120,-52.853,-179.718,6.559,149.117
C00724=1136.533,64.369,-52.869,-179.715,6.559,149.116
C00725=1136.528,64.619,-52.885,-179.713,6.561,149.116
C00726=1136.523,64.868,-52.901,-179.710,6.562,149.115
C00727=1136.519,65.118,-52.918,-179.708,6.563,149.115
C00728=1136.514,65.368,-52.934,-179.705,6.565,149.114
C00729=1136.508,65.617,-52.951,-179.702,6.566,149.114
C00730=1136.504,65.866,-52.967,-179.700,6.567,149.114
C00731=1136.498,66.116,-52.983,-179.697,6.569,149.113
C00732=1136.494,66.365,-53.000,-179.694,6.570,149.112
C00733=1136.489,66.614,-53.016,-179.692,6.571,149.112
C00734=1136.484,66.864,-53.032,-179.689,6.572,149.112
C00735=1136.479,67.113,-53.048,-179.686,6.574,149.111
C00736=1136.474,67.363,-53.066,-179.683,6.575,149.110
C00737=1136.468,67.611,-53.082,-179.681,6.576,149.110
C00738=1136.464,67.861,-53.098,-179.678,6.578,149.110
C00739=1136.459,68.111,-53.114,-179.675,6.580,149.109
C00740=1136.454,68.360,-53.131,-179.672,6.580,149.108
C00741=1136.449,68.610,-53.148,-179.670,6.582,149.108
C00742=1136.444,68.859,-53.164,-179.667,6.583,149.108
C00743=1136.439,69.108,-53.180,-179.665,6.584,149.107
C00744=1136.435,69.358,-53.197,-179.662,6.585,149.107
C00745=1136.429,69.607,-53.214,-179.659,6.587,149.106
C00746=1136.424,69.856,-53.231,-179.657,6.588,149.106
C00747=1136.419,70.106,-53.246,-179.654,6.590,149.105
C00748=1136.414,70.355,-53.263,-179.651,6.591,149.105
C00749=1136.409,70.605,-53.280,-179.648,6.592,149.104
C00750=1136.404,70.854,-53.296,-179.646,6.593,149.104
C00751=1136.400,71.103,-53.313,-179.643,6.595,149.103
C00752=1136.394,71.353,-53.330,-179.640,6.596,149.103
C00753=1136.389,71.602,-53.347,-179.638,6.597,149.102
C00754=1136.385,71.852,-53.363,-179.635,6.599,149.102
C00755=1136.379,72.101,-53.379,-179.632,6.600,149.101
C00756=1136.374,72.351,-53.396,-179.629,6.602,149.101
C00757=1136.370,72.600,-53.413,-179.627,6.603,149.100
C00758=1136.364,72.849,-53.430,-179.624,6.604,149.100
C00759=1136.359,73.099,-53.446,-179.621,6.606,149.099
C00760=1136.355,73.348,-53.463,-179.618,6.607,149.099
C00761=1136.349,73.597,-53.480,-179.616,6.608,149.098
C00762=1136.345,73.847,-53.497,-179.613,6.610,149.098
C00763=1136.340,74.096,-53.513,-179.610,6.611,149.097
C00764=1136.335,74.346,-53.530,-179.607,6.613,149.097
C00765=1136.330,74.595,-53.547,-179.605,6.613,149.096
C00766=1136.325,74.845,-53.564,-179.602,6.615,149.096
C00767=1136.320,75.094,-53.581,-179.600,6.617,149.095
C00768=1136.315,75.343,-53.597,-179.597,6.618,149.095
C00769=1136.310,75.593,-53.614,-179.594,6.619,149.094
C00770=1136.305,75.842,-53.631,-179.591,6.620,149.094
C00771=1136.300,76.092,-53.648,-179.589,6.622,149.094
C00772=1136.295,76.341,-53.665,-179.586,6.624,149.093
C00773=1136.290,76.590,-53.683,-179.583,6.624,149.092
C00774=1136.286,76.839,-53.699,-179.581,6.626,149.092
C00775=1136.280,77.089,-53.716,-179.578,6.628,149.092
C00776=1136.275,77.338,-53.733,-179.575,6.629,149.091
C00777=1136.270,77.588,-53.750,-179.573,6.630,149.091
C00778=1136.266,77.837,-53.767,-179.570,6.631,149.090
C00779=1136.261,78.087,-53.784,-179.567,6.633,149.090
C00780=1136.255,78.336,-53.800,-179.564,6.635,149.089
C00781=1136.251,78.585,-53.818,-179.562,6.636,149.089
C00782=1136.246,78.835,-53.835,-179.559,6.637,149.088
C00783=1136.240,79.103,-53.853,-179.556,6.638,149.088
C00784=1136.235,79.371,-53.871,-179.553,6.640,149.087
C00785=1136.230,79.640,-53.890,-179.550,6.641,149.087
C00786=1136.225,79.908,-53.908,-179.547,6.643,149.086
C00787=1136.220,80.158,-53.925,-179.545,6.645,149.086
C00788=1136.215,80.407,-53.943,-179.542,6.646,149.085
C00789=1136.210,80.656,-53.960,-179.539,6.648,149.085
C00790=1136.204,80.906,-53.977,-179.536,6.649,149.084
C00791=1136.200,81.154,-53.994,-179.534,6.650,149.084
C00792=1136.195,81.404,-54.011,-179.531,6.652,149.083
C00793=1136.190,81.654,-54.028,-179.528,6.653,149.083
C00794=1136.185,81.904,-54.045,-179.526,6.654,149.082
C00795=1136.180,82.153,-54.063,-179.523,6.656,149.082
C00796=1136.175,82.401,-54.079,-179.520,6.657,149.081
C00797=1136.170,82.651,-54.097,-179.517,6.659,149.081
C00798=1136.165,82.900,-54.115,-179.514,6.660,149.080
C00799=1136.161,83.150,-54.131,-179.512,6.661,149.080
C00800=1136.156,83.399,-54.149,-179.509,6.663,149.080
C00801=1136.151,83.649,-54.167,-179.507,6.664,149.079
C00802=1136.146,83.898,-54.183,-179.504,6.666,149.079
C00803=1136.141,84.147,-54.201,-179.501,6.668,149.078
C00804=1136.135,84.397,-54.218,-179.498,6.669,149.078
C00805=1136.131,84.646,-54.236,-179.496,6.670,149.077
C00806=1136.126,84.895,-54.253,-179.493,6.672,149.077
C00807=1136.121,85.144,-54.271,-179.490,6.673,149.076
C00808=1136.117,85.394,-54.287,-179.487,6.675,149.076
C00809=1136.111,85.644,-54.305,-179.484,6.676,149.075
C00810=1136.106,85.893,-54.323,-179.481,6.678,149.075
C00811=1136.102,86.142,-54.339,-179.479,6.679,149.074
C00812=1136.097,86.392,-54.357,-179.477,6.680,149.074
C00813=1136.092,86.641,-54.375,-179.474,6.682,149.074
C00814=1136.086,86.890,-54.392,-179.471,6.683,149.073
C00815=1136.082,87.139,-54.410,-179.468,6.685,149.072
C00816=1136.077,87.389,-54.427,-179.465,6.687,149.072
C00817=1136.072,87.638,-54.445,-179.463,6.687,149.072
C00818=1136.067,87.887,-54.462,-179.460,6.689,149.071
C00819=1136.062,88.137,-54.480,-179.457,6.691,149.071
C00820=1136.057,88.386,-54.497,-179.454,6.692,149.070
C00821=1136.052,88.635,-54.515,-179.452,6.694,149.070
C00822=1136.048,88.885,-54.533,-179.449,6.695,149.069
C00823=1136.042,89.134,-54.550,-179.447,6.696,149.069
C00824=1136.037,89.383,-54.568,-179.444,6.698,149.068
C00825=1136.033,89.632,-54.585,-179.441,6.700,149.068
C00826=1136.028,89.882,-54.603,-179.438,6.701,149.067
C00827=1136.023,90.131,-54.621,-179.435,6.703,149.067
C00828=1136.018,90.380,-54.639,-179.432,6.704,149.067
C00829=1136.013,90.630,-54.656,-179.430,6.706,149.066
C00830=1136.008,90.879,-54.674,-179.428,6.707,149.066
C00831=1136.003,91.129,-54.692,-179.425,6.708,149.065
C00832=1135.999,91.378,-54.708,-179.422,6.710,149.065
C00833=1135.994,91.627,-54.726,-179.419,6.711,149.064
C00834=1135.989,91.876,-54.744,-179.416,6.713,149.064
C00835=1135.984,92.126,-54.762,-179.413,6.715,149.063
C00836=1135.979,92.375,-54.780,-179.411,6.716,149.063
C00837=1135.974,92.625,-54.798,-179.408,6.718,149.063
C00838=1135.969,92.874,-54.816,-179.405,6.719,149.062
C00839=1135.964,93.123,-54.834,-179.403,6.720,149.061
C00840=1135.959,93.372,-54.852,-179.400,6.722,149.061
C00841=1135.954,93.622,-54.869,-179.397,6.724,149.061
C00842=1135.949,93.871,-54.887,-179.394,6.725,149.060
C00843=1135.945,94.121,-54.905,-179.392,6.727,149.060
C00844=1135.940,94.370,-54.923,-179.389,6.729,149.059
C00845=1135.935,94.619,-54.941,-179.386,6.730,149.059
C00846=1135.930,94.869,-54.959,-179.383,6.731,149.058
C00847=1135.925,95.118,-54.976,-179.380,6.733,149.058
C00848=1135.920,95.367,-54.994,-179.378,6.734,149.057
C00849=1135.915,95.617,-55.012,-179.375,6.736,149.057
C00850=1135.910,95.866,-55.030,-179.372,6.737,149.057
C00851=1135.905,96.115,-55.048,-179.369,6.739,149.056
C00852=1135.900,96.364,-55.066,-179.367,6.740,149.056
C00853=1135.895,96.613,-55.084,-179.364,6.742,149.055
C00854=1135.891,96.863,-55.103,-179.361,6.744,149.055
C00855=1135.886,97.112,-55.121,-179.358,6.745,149.054
C00856=1135.881,97.362,-55.139,-179.356,6.747,149.054
C00857=1135.876,97.611,-55.157,-179.353,6.749,149.053
C00858=1135.871,97.860,-55.175,-179.350,6.750,149.053
C00859=1135.866,98.109,-55.192,-179.347,6.751,149.052
C00860=1135.861,98.358,-55.210,-179.345,6.753,149.052
C00861=1135.857,98.608,-55.229,-179.342,6.754,149.052
C00862=1135.852,98.857,-55.247,-179.339,6.756,149.051
C00863=1135.847,99.107,-55.265,-179.337,6.758,149.051
C00864=1135.842,99.356,-55.283,-179.334,6.759,149.050
C00865=1135.837,99.605,-55.301,-179.331,6.761,149.050
C00866=1135.832,99.854,-55.319,-179.328,6.763,149.049
C00867=1135.828,100.104,-55.338,-179.325,6.764,149.049
C00868=1135.823,100.353,-55.356,-179.322,6.765,149.048
C00869=1135.818,100.602,-55.374,-179.320,6.767,149.048
C00870=1135.813,100.851,-55.392,-179.317,6.769,149.048
C00871=1135.807,101.101,-55.411,-179.314,6.771,149.047
C00872=1135.803,101.351,-55.429,-179.311,6.772,149.047
C00873=1135.798,101.600,-55.447,-179.309,6.774,149.046
C00874=1135.793,101.849,-55.465,-179.306,6.776,149.046
C00875=1135.789,102.097,-55.484,-179.303,6.777,149.045
C00876=1135.784,102.348,-55.503,-179.301,6.778,149.045
C00877=1135.779,102.597,-55.521,-179.298,6.779,149.044
C00878=1135.774,102.846,-55.539,-179.295,6.781,149.044
C00879=1135.769,103.095,-55.557,-179.292,6.783,149.044
C00880=1135.764,103.344,-55.575,-179.290,6.784,149.043
C00881=1135.759,103.594,-55.594,-179.287,6.786,149.043
C00882=1135.754,103.843,-55.612,-179.284,6.788,149.042
C00883=1135.749,104.092,-55.630,-179.281,6.789,149.042
C00884=1135.745,104.341,-55.649,-179.279,6.791,149.042
C00885=1135.740,104.591,-55.668,-179.275,6.792,149.041
C00886=1135.735,104.840,-55.686,-179.273,6.794,149.041
C00887=1135.730,105.108,-55.705,-179.270,6.796,149.040
C00888=1135.724,105.376,-55.726,-179.267,6.798,149.040
C00889=1135.720,105.645,-55.746,-179.264,6.800,149.039
C00890=1135.714,105.914,-55.766,-179.261,6.801,149.039
C00891=1135.709,106.162,-55.785,-179.258,6.803,149.038
C00892=1135.704,106.412,-55.803,-179.255,6.805,149.038
C00893=1135.699,106.662,-55.822,-179.253,6.806,149.037
C00894=1135.695,106.910,-55.840,-179.250,6.808,149.037
C00895=1135.689,107.160,-55.859,-179.247,6.810,149.037
C00896=1135.685,107.409,-55.878,-179.244,6.811,149.036
C00897=1135.680,107.658,-55.896,-179.242,6.813,149.036
C00898=1135.675,107.908,-55.914,-179.239,6.815,149.035
C00899=1135.671,108.157,-55.933,-179.236,6.816,149.035
C00900=1135.666,108.406,-55.951,-179.233,6.818,149.035
C00901=1135.661,108.656,-55.971,-179.230,6.819,149.034
C00902=1135.656,108.905,-55.989,-179.227,6.821,149.033
C00903=1135.651,109.154,-56.008,-179.225,6.823,149.033
C00904=1135.646,109.404,-56.027,-179.222,6.824,149.033
C00905=1135.642,109.652,-56.045,-179.219,6.826,149.032
C00906=1135.636,109.902,-56.064,-179.217,6.828,149.032
C00907=1135.632,110.151,-56.083,-179.214,6.829,149.031
C00908=1135.626,110.400,-56.102,-179.211,6.831,149.031
C00909=1135.622,110.650,-56.121,-179.208,6.833,149.031
C00910=1135.617,110.899,-56.140,-179.206,6.834,149.030
C00911=1135.612,111.148,-56.158,-179.203,6.836,149.030
C00912=1135.607,111.397,-56.178,-179.200,6.838,149.029
C00913=1135.603,111.647,-56.196,-179.197,6.839,149.029
C00914=1135.598,111.896,-56.215,-179.195,6.841,149.029
C00915=1135.593,112.145,-56.234,-179.192,6.843,149.028
C00916=1135.588,112.394,-56.253,-179.189,6.844,149.028
C00917=1135.584,112.643,-56.272,-179.186,6.846,149.027
C00918=1135.578,112.892,-56.291,-179.183,6.847,149.027
C00919=1135.574,113.142,-56.309,-179.181,6.849,149.026
C00920=1135.569,113.391,-56.328,-179.178,6.851,149.026
C00921=1135.565,113.640,-56.348,-179.175,6.852,149.026
C00922=1135.559,113.890,-56.366,-179.172,6.854,149.025
C00923=1135.554,114.139,-56.385,-179.169,6.857,149.025
C00924=1135.550,114.388,-56.404,-179.166,6.858,149.024
C00925=1135.544,114.637,-56.423,-179.164,6.860,149.024
C00926=1135.540,114.887,-56.442,-179.161,6.862,149.023
C00927=1135.535,115.135,-56.461,-179.158,6.863,149.023
C00928=1135.530,115.385,-56.480,-179.155,6.865,149.023
C00929=1135.525,115.634,-56.500,-179.153,6.867,149.022
C00930=1135.520,115.884,-56.519,-179.150,6.868,149.022
C00931=1135.516,116.132,-56.537,-179.147,6.870,149.021
C00932=1135.511,116.382,-56.557,-179.144,6.872,149.021
C00933=1135.505,116.631,-56.576,-179.142,6.873,149.021
C00934=1135.501,116.880,-56.595,-179.139,6.875,149.020
C00935=1135.496,117.130,-56.614,-179.136,6.877,149.020
C00936=1135.491,117.379,-56.634,-179.134,6.878,149.019
C00937=1135.486,117.628,-56.652,-179.131,6.880,149.019
C00938=1135.482,117.877,-56.672,-179.128,6.882,149.019
C00939=1135.476,118.126,-56.691,-179.125,6.884,149.018
C00940=1135.472,118.375,-56.710,-179.122,6.886,149.018
C00941=1135.468,118.625,-56.730,-179.119,6.888,149.017
C00942=1135.462,118.874,-56.749,-179.117,6.889,149.017
C00943=1135.458,119.123,-56.768,-179.114,6.891,149.017
C00944=1135.453,119.372,-56.788,-179.111,6.893,149.016
C00945=1135.448,119.621,-56.807,-179.108,6.894,149.016
C00946=1135.443,119.870,-56.827,-179.105,6.896,149.015
C00947=1135.439,120.120,-56.846,-179.102,6.897,149.015
C00948=1135.434,120.369,-56.865,-179.100,6.899,149.014
C00949=1135.429,120.618,-56.885,-179.097,6.901,149.014
C00950=1135.424,120.868,-56.904,-179.094,6.903,149.014
C00951=1135.419,121.116,-56.923,-179.091,6.905,149.013
C00952=1135.415,121.366,-56.943,-179.088,6.907,149.013
C00953=1135.410,121.615,-56.962,-179.085,6.908,149.012
C00954=1135.405,121.864,-56.982,-179.083,6.910,149.012
C00955=1135.400,122.114,-57.001,-179.080,6.912,149.012
C00956=1135.395,122.362,-57.020,-179.077,6.913,149.011
C00957=1135.390,122.612,-57.040,-179.075,6.915,149.011
C00958=1135.386,122.861,-57.059,-179.072,6.917,149.010
C00959=1135.380,123.110,-57.079,-179.068,6.919,149.010
C00960=1135.376,123.360,-57.098,-179.066,6.921,149.010
C00961=1135.371,123.609,-57.119,-179.063,6.923,149.009
C00962=1135.366,123.858,-57.138,-179.061,6.925,149.009
C00963=1135.362,124.107,-57.157,-179.058,6.926,149.009
C00964=1135.357,124.356,-57.177,-179.055,6.928,149.008
C00965=1135.352,124.605,-57.196,-179.053,6.930,149.008
C00966=1135.347,124.854,-57.216,-179.050,6.931,149.007
C00967=1135.343,125.104,-57.236,-179.047,6.934,149.007
C00968=1135.337,125.353,-57.255,-179.044,6.936,149.007
C00969=1135.332,125.602,-57.275,-179.041,6.937,149.006
C00970=1135.328,125.852,-57.294,-179.038,6.939,149.006
C00971=1135.323,126.101,-57.315,-179.036,6.941,149.005
C00972=1135.318,126.350,-57.334,-179.033,6.942,149.005
C00973=1135.314,126.599,-57.353,-179.030,6.944,149.005
C00974=1135.309,126.848,-57.374,-179.027,6.947,149.004
C00975=1135.304,127.097,-57.393,-179.024,6.948,149.004
C00976=1135.299,127.346,-57.413,-179.021,6.950,149.003
C00977=1135.295,127.595,-57.433,-179.019,6.952,149.003
C00978=1135.290,127.845,-57.453,-179.016,6.953,149.003
C00979=1135.285,128.094,-57.472,-179.013,6.955,149.002
C00980=1135.280,128.343,-57.492,-179.010,6.957,149.002
C00981=1135.276,128.592,-57.512,-179.007,6.959,149.001
C00982=1135.271,128.842,-57.532,-179.004,6.961,149.001
C00983=1135.266,129.090,-57.552,-179.002,6.963,149.001
C00984=1135.261,129.340,-57.571,-178.999,6.964,149.000
C00985=1135.257,129.589,-57.592,-178.996,6.966,149.000
C00986=1135.251,129.838,-57.612,-178.993,6.968,148.999
C00987=1135.246,130.087,-57.631,-178.990,6.970,148.999
C00988=1135.241,130.336,-57.651,-178.988,6.972,148.999
C00989=1135.237,130.586,-57.671,-178.985,6.973,148.998
C00990=1135.232,130.835,-57.691,-178.983,6.976,148.998
C00991=1135.227,131.103,-57.713,-178.979,6.978,148.997
C00992=1135.222,131.372,-57.734,-178.976,6.979,148.997
C00993=1135.217,131.640,-57.756,-178.973,6.982,148.997
C00994=1135.211,131.909,-57.778,-178.970,6.984,148.996
C00995=1135.207,132.158,-57.798,-178.967,6.985,148.996
C00996=1135.202,132.407,-57.817,-178.965,6.987,148.995
C00997=1135.197,132.656,-57.838,-178.961,6.989,148.995
C00998=1135.193,132.906,-57.857,-178.959,6.991,148.995
C00999=1135.188,133.155,-57.878,-178.956,6.993,148.994
C01000=1135.184,133.404,-57.898,-178.954,6.995,148.994
C01001=1135.178,133.653,-57.918,-178.951,6.997,148.994
C01002=1135.173,133.902,-57.938,-178.948,6.999,148.993
C01003=1135.168,134.151,-57.958,-178.945,7.001,148.993
C01004=1135.164,134.400,-57.978,-178.942,7.002,148.993
C01005=1135.160,134.649,-57.999,-178.939,7.004,148.992
C01006=1135.154,134.899,-58.019,-178.937,7.006,148.992
C01007=1135.150,135.148,-58.039,-178.933,7.008,148.991
C01008=1135.145,135.397,-58.060,-178.931,7.010,148.991
C01009=1135.140,135.647,-58.079,-178.928,7.012,148.991
C01010=1135.135,135.895,-58.100,-178.925,7.013,148.990
C01011=1135.130,136.144,-58.120,-178.922,7.016,148.990
C01012=1135.126,136.393,-58.141,-178.920,7.018,148.990
C01013=1135.121,136.643,-58.160,-178.917,7.020,148.989
C01014=1135.116,136.892,-58.181,-178.914,7.021,148.989
C01015=1135.111,137.141,-58.202,-178.911,7.023,148.988
C01016=1135.107,137.390,-58.222,-178.908,7.026,148.988
C01017=1135.103,137.639,-58.243,-178.905,7.027,148.988
C01018=1135.097,137.889,-58.263,-178.903,7.029,148.987
C01019=1135.093,138.138,-58.283,-178.900,7.031,148.987
C01020=1135.088,138.386,-58.304,-178.897,7.033,148.987
C01021=1135.083,138.636,-58.325,-178.894,7.035,148.986
C01022=1135.079,138.885,-58.345,-178.892,7.037,148.986
C01023=1135.074,139.134,-58.365,-178.889,7.039,148.986
C01024=1135.069,139.383,-58.386,-178.886,7.041,148.985
C01025=1135.064,139.632,-58.406,-178.883,7.043,148.985
C01026=1135.060,139.881,-58.426,-178.880,7.044,148.984
C01027=1135.055,140.131,-58.447,-178.877,7.046,148.984
C01028=1135.050,140.380,-58.468,-178.874,7.049,148.984
C01029=1135.045,140.629,-58.489,-178.871,7.050,148.983
C01030=1135.041,140.878,-58.509,-178.869,7.052,148.983
C01031=1135.036,141.127,-58.529,-178.866,7.054,148.983
C01032=1135.031,141.376,-58.550,-178.863,7.057,148.982
C01033=1135.026,141.625,-58.571,-178.860,7.058,148.982
C01034=1135.021,141.874,-58.592,-178.858,7.060,148.982
C01035=1135.017,142.123,-58.612,-178.854,7.063,148.981
C01036=1135.012,142.372,-58.632,-178.852,7.064,148.981
C01037=1135.007,142.621,-58.653,-178.849,7.066,148.981
C01038=1135.003,142.870,-58.674,-178.847,7.068,148.980
C01039=1134.998,143.120,-58.695,-178.843,7.070,148.980
C01040=1134.993,143.369,-58.715,-178.841,7.072,148.979
C01041=1134.988,143.618,-58.736,-178.838,7.074,148.979
C01042=1134.984,143.867,-58.756,-178.835,7.076,148.979
C01043=1134.978,144.116,-58.777,-178.832,7.078,148.978
C01044=1134.974,144.364,-58.798,-178.830,7.080,148.978
C01045=1134.969,144.614,-58.819,-178.827,7.082,148.978
C01046=1134.965,144.863,-58.840,-178.824,7.084,148.977
C01047=1134.960,145.113,-58.861,-178.821,7.086,148.977
C01048=1134.956,145.361,-58.881,-178.818,7.088,148.977
C01049=1134.951,145.611,-58.902,-178.815,7.090,148.976
C01050=1134.945,145.860,-58.923,-178.813,7.092,148.976
C01051=1134.941,146.108,-58.944,-178.810,7.094,148.976
C01052=1134.936,146.358,-58.965,-178.807,7.096,148.975
C01053=1134.932,146.607,-58.986,-178.804,7.098,148.975
C01054=1134.926,146.856,-59.007,-178.801,7.100,148.975
C01055=1134.922,147.104,-59.028,-178.799,7.102,148.974
C01056=1134.918,147.354,-59.049,-178.796,7.105,148.974
C01057=1134.913,147.603,-59.070,-178.793,7.106,148.974
C01058=1134.908,147.852,-59.091,-178.790,7.108,148.973
C01059=1134.903,148.101,-59.112,-178.787,7.110,148.973
C01060=1134.898,148.350,-59.133,-178.784,7.112,148.972
C01061=1134.894,148.599,-59.154,-178.781,7.114,148.972
C01062=1134.889,148.848,-59.175,-178.779,7.117,148.972
C01063=1134.884,149.098,-59.197,-178.776,7.118,148.972
C01064=1134.880,149.347,-59.217,-178.773,7.120,148.971
C01065=1134.875,149.595,-59.239,-178.770,7.123,148.971
C01066=1134.870,149.845,-59.260,-178.767,7.124,148.970
C01067=1134.865,150.094,-59.280,-178.765,7.126,148.970
C01068=1134.861,150.343,-59.302,-178.762,7.129,148.970
C01069=1134.856,150.592,-59.323,-178.759,7.131,148.969
C01070=1134.852,150.840,-59.344,-178.756,7.132,148.969
C01071=1134.847,151.090,-59.365,-178.753,7.135,148.969
C01072=1134.842,151.338,-59.387,-178.751,7.137,148.969
C01073=1134.837,151.588,-59.408,-178.748,7.139,148.968
C01074=1134.833,151.837,-59.428,-178.745,7.141,148.968
C01075=1134.828,152.086,-59.450,-178.742,7.143,148.967
C01076=1134.823,152.335,-59.471,-178.739,7.144,148.967
C01077=1134.818,152.584,-59.493,-178.736,7.147,148.967
C01078=1134.813,152.834,-59.514,-178.734,7.149,148.967
C01079=1134.809,153.082,-59.535,-178.731,7.151,148.966
C01080=1134.804,153.331,-59.557,-178.728,7.153,148.966
C01081=1134.800,153.581,-59.578,-178.725,7.155,148.965
C01082=1134.795,153.829,-59.600,-178.722,7.158,148.965
C01083=1134.790,154.079,-59.621,-178.719,7.160,148.965
C01084=1134.785,154.327,-59.643,-178.717,7.161,148.964
C01085=1134.781,154.577,-59.663,-178.713,7.164,148.964
C01086=1134.776,154.826,-59.685,-178.711,7.166,148.964
C01087=1134.771,155.074,-59.707,-178.708,7.168,148.964
C01088=1134.766,155.324,-59.728,-178.705,7.170,148.963
C01089=1134.762,155.573,-59.750,-178.702,7.172,148.963
C01090=1134.757,155.821,-59.771,-178.700,7.175,148.963
C01091=1134.752,156.071,-59.793,-178.697,7.176,148.962
C01092=1134.748,156.320,-59.814,-178.694,7.178,148.962
C01093=1134.743,156.568,-59.835,-178.691,7.181,148.962
C01094=1134.738,156.818,-59.856,-178.689,7.183,148.961
C01095=1134.733,157.086,-59.880,-178.685,7.185,148.961
C01096=1134.728,157.355,-59.903,-178.683,7.187,148.961
C01097=1134.723,157.625,-59.927,-178.679,7.189,148.960
C01098=1134.718,157.893,-59.950,-178.676,7.192,148.960
C01099=1134.714,158.143,-59.972,-178.673,7.194,148.960
C01100=1134.709,158.392,-59.993,-178.670,7.196,148.959
C01101=1134.704,158.640,-60.015,-178.668,7.198,148.959
C01102=1134.700,158.890,-60.037,-178.665,7.200,148.959
C01103=1134.695,159.138,-60.059,-178.662,7.202,148.958
C01104=1134.690,159.388,-60.081,-178.659,7.204,148.958
C01105=1134.685,159.637,-60.102,-178.656,7.207,148.958
C01106=1134.680,159.886,-60.123,-178.653,7.209,148.957
C01107=1134.676,160.135,-60.145,-178.651,7.210,148.957
C01108=1134.671,160.384,-60.167,-178.648,7.213,148.957
C01109=1134.667,160.633,-60.189,-178.645,7.215,148.956
C01110=1134.662,160.882,-60.211,-178.642,7.217,148.956
C01111=1134.657,161.131,-60.233,-178.639,7.219,148.956
C01112=1134.652,161.380,-60.255,-178.636,7.222,148.956
C01113=1134.647,161.629,-60.277,-178.634,7.224,148.955
C01114=1134.643,161.878,-60.299,-178.631,7.225,148.955
C01115=1134.638,162.127,-60.320,-178.628,7.228,148.955
C01116=1134.634,162.376,-60.342,-178.625,7.230,148.954
C01117=1134.629,162.624,-60.364,-178.622,7.233,148.954
C01118=1134.625,162.874,-60.386,-178.620,7.235,148.954
C01119=1134.620,163.122,-60.408,-178.617,7.237,148.953
C01120=1134.616,163.372,-60.430,-178.614,7.239,148.953
C01121=1134.611,163.620,-60.452,-178.611,7.241,148.953
C01122=1134.606,163.870,-60.474,-178.608,7.243,148.953
C01123=1134.601,164.119,-60.496,-178.606,7.245,148.952
C01124=1134.597,164.368,-60.518,-178.602,7.248,148.952
C01125=1134.592,164.617,-60.540,-178.600,7.250,148.952
C01126=1134.588,164.866,-60.562,-178.597,7.252,148.951
C01127=1134.583,165.115,-60.583,-178.594,7.254,148.951
C01128=1134.578,165.364,-60.606,-178.591,7.257,148.951
C01129=1134.573,165.612,-60.628,-178.588,7.259,148.950
C01130=1134.569,165.862,-60.650,-178.585,7.261,148.950
C01131=1134.564,166.110,-60.672,-178.583,7.263,148.950
C01132=1134.559,166.360,-60.695,-178.580,7.266,148.950
C01133=1134.554,166.609,-60.716,-178.577,7.267,148.949
C01134=1134.550,166.858,-60.739,-178.574,7.270,148.949
C01135=1134.545,167.106,-60.761,-178.571,7.272,148.949
C01136=1134.540,167.356,-60.784,-178.569,7.274,148.948
C01137=1134.535,167.604,-60.805,-178.566,7.277,148.948
C01138=1134.531,167.854,-60.827,-178.563,7.278,148.948
C01139=1134.527,168.102,-60.850,-178.560,7.281,148.947
C01140=1134.522,168.351,-60.872,-178.558,7.283,148.947
C01141=1134.517,168.601,-60.894,-178.554,7.285,148.947
C01142=1134.513,168.849,-60.917,-178.552,7.287,148.947
C01143=1134.508,169.098,-60.939,-178.549,7.290,148.946
C01144=1134.503,169.347,-60.961,-178.546,7.292,148.946
C01145=1134.499,169.596,-60.984,-178.543,7.294,148.946
C01146=1134.494,169.845,-61.007,-178.541,7.296,148.946
C01147=1134.489,170.094,-61.028,-178.537,7.299,148.945
C01148=1134.485,170.343,-61.051,-178.535,7.301,148.945
C01149=1134.480,170.592,-61.074,-178.532,7.303,148.945
C01150=1134.475,170.841,-61.095,-178.529,7.305,148.944
C01151=1134.470,171.090,-61.119,-178.526,7.308,148.944
C01152=1134.466,171.339,-61.140,-178.523,7.310,148.944
C01153=1134.462,171.587,-61.163,-178.520,7.312,148.943
C01154=1134.457,171.837,-61.186,-178.518,7.314,148.943
C01155=1134.452,172.085,-61.208,-178.515,7.317,148.943
C01156=1134.447,172.335,-61.231,-178.512,7.319,148.943
C01157=1134.443,172.583,-61.254,-178.509,7.321,148.942
C01158=1134.438,172.832,-61.276,-178.506,7.323,148.942
C01159=1134.434,173.081,-61.299,-178.503,7.326,148.942
C01160=1134.429,173.330,-61.321,-178.500,7.329,148.942
C01161=1134.424,173.579,-61.344,-178.498,7.330,148.941
C01162=1134.420,173.828,-61.366,-178.495,7.333,148.941
C01163=1134.415,174.077,-61.389,-178.492,7.335,148.941
C01164=1134.411,174.327,-61.411,-178.489,7.337,148.940
C01165=1134.405,174.575,-61.434,-178.487,7.340,148.940
C01166=1134.401,174.824,-61.457,-178.483,7.342,148.940
C01167=1134.396,175.073,-61.479,-178.481,7.344,148.940
C01168=1134.392,175.321,-61.502,-178.478,7.347,148.939
C01169=1134.387,175.571,-61.525,-178.475,7.348,148.939
C01170=1134.383,175.820,-61.547,-178.472,7.351,148.939
C01171=1134.378,176.069,-61.571,-178.469,7.353,148.939
C01172=1134.373,176.318,-61.593,-178.467,7.356,148.938
C01173=1134.369,176.566,-61.616,-178.463,7.358,148.938
C01174=1134.364,176.815,-61.639,-178.461,7.360,148.938
C01175=1134.360,177.064,-61.662,-178.458,7.363,148.938
C01176=1134.354,177.313,-61.684,-178.455,7.365,148.937
C01177=1134.350,177.562,-61.707,-178.452,7.368,148.937
C01178=1134.346,177.811,-61.730,-178.450,7.369,148.937
C01179=1134.341,178.060,-61.754,-178.447,7.372,148.937
C01180=1134.337,178.309,-61.776,-178.444,7.374,148.936
C01181=1134.331,178.557,-61.799,-178.441,7.376,148.936
C01182=1134.327,178.806,-61.822,-178.438,7.379,148.936
C01183=1134.323,179.055,-61.845,-178.435,7.381,148.935
C01184=1134.318,179.304,-61.868,-178.432,7.384,148.935
C01185=1134.313,179.554,-61.891,-178.430,7.386,148.935
C01186=1134.309,179.802,-61.913,-178.427,7.388,148.935
C01187=1134.304,180.051,-61.937,-178.424,7.391,148.934
C01188=1134.299,180.300,-61.960,-178.421,7.393,148.934
C01189=1134.295,180.549,-61.983,-178.418,7.396,148.934
C01190=1134.290,180.798,-62.006,-178.415,7.397,148.934
C01191=1134.286,181.047,-62.029,-178.413,7.400,148.933
C01192=1134.282,181.295,-62.052,-178.410,7.402,148.933
C01193=1134.277,181.544,-62.075,-178.407,7.405,148.933
C01194=1134.272,181.793,-62.098,-178.404,7.407,148.933
C01195=1134.267,182.042,-62.122,-178.401,7.409,148.932
C01196=1134.263,182.291,-62.144,-178.398,7.412,148.932
C01197=1134.258,182.540,-62.167,-178.396,7.414,148.932
C01198=1134.253,182.789,-62.191,-178.393,7.417,148.932
C01199=1134.248,183.058,-62.216,-178.390,7.419,148.931
C01200=1134.243,183.328,-62.241,-178.387,7.422,148.931
C01201=1134.239,183.598,-62.266,-178.383,7.425,148.931
C01202=1134.234,183.867,-62.292,-178.380,7.427,148.931
C01203=1134.229,184.116,-62.315,-178.378,7.429,148.930
C01204=1134.224,184.365,-62.338,-178.375,7.432,148.930
C01205=1134.219,184.614,-62.362,-178.372,7.435,148.930
C01206=1134.215,184.863,-62.385,-178.369,7.437,148.930
C01207=1134.211,185.112,-62.408,-178.366,7.439,148.929
C01208=1134.206,185.361,-62.431,-178.364,7.441,148.929
C01209=1134.201,185.610,-62.454,-178.361,7.444,148.929
C01210=1134.197,185.859,-62.478,-178.358,7.447,148.929
C01211=1134.192,186.107,-62.502,-178.355,7.448,148.928
C01212=1134.188,186.356,-62.525,-178.352,7.451,148.928
C01213=1134.183,186.605,-62.549,-178.349,7.454,148.928
C01214=1134.178,186.854,-62.572,-178.347,7.456,148.928
C01215=1134.173,187.103,-62.595,-178.343,7.458,148.927
C01216=1134.170,187.351,-62.619,-178.341,7.460,148.927
C01217=1134.165,187.600,-62.642,-178.338,7.463,148.927
C01218=1134.160,187.849,-62.666,-178.335,7.466,148.927
C01219=1134.156,188.098,-62.690,-178.332,7.468,148.926
C01220=1134.151,188.347,-62.713,-178.330,7.471,148.926
C01221=1134.147,188.596,-62.736,-178.326,7.473,148.926
C01222=1134.142,188.845,-62.760,-178.324,7.475,148.926
C01223=1134.138,189.093,-62.784,-178.321,7.478,148.926
C01224=1134.133,189.342,-62.807,-178.318,7.481,148.925
C01225=1134.128,189.591,-62.830,-178.315,7.482,148.925
C01226=1134.124,189.840,-62.855,-178.312,7.485,148.925
C01227=1134.119,190.089,-62.878,-178.309,7.488,148.925
C01228=1134.115,190.337,-62.902,-178.307,7.490,148.924
C01229=1134.110,190.586,-62.925,-178.304,7.493,148.924
C01230=1134.104,190.836,-62.949,-178.301,7.495,148.924
C01231=1134.100,191.084,-62.973,-178.299,7.497,148.924
C01232=1134.095,191.333,-62.997,-178.295,7.500,148.924
C01233=1134.091,191.582,-63.021,-178.292,7.503,148.923
C01234=1134.086,191.831,-63.044,-178.290,7.504,148.923
C01235=1134.082,192.079,-63.068,-178.287,7.507,148.923
C01236=1134.077,192.328,-63.092,-178.284,7.510,148.923
C01237=1134.073,192.577,-63.116,-178.281,7.512,148.922
C01238=1134.069,192.826,-63.139,-178.279,7.515,148.922
C01239=1134.064,193.075,-63.163,-178.275,7.517,148.922
C01240=1134.059,193.324,-63.187,-178.273,7.519,148.922
C01241=1134.054,193.572,-63.212,-178.270,7.522,148.922
C01242=1134.050,193.821,-63.235,-178.267,7.525,148.921
C01243=1134.045,194.070,-63.259,-178.264,7.527,148.921
C01244=1134.041,194.318,-63.283,-178.261,7.529,148.921
C01245=1134.037,194.568,-63.307,-178.259,7.532,148.921
C01246=1134.032,194.817,-63.331,-178.255,7.535,148.920
C01247=1134.027,195.066,-63.355,-178.253,7.537,148.920
C01248=1134.023,195.314,-63.379,-178.250,7.540,148.920
C01249=1134.018,195.562,-63.403,-178.247,7.542,148.920
C01250=1134.014,195.812,-63.426,-178.245,7.544,148.920
C01251=1134.009,196.061,-63.451,-178.241,7.547,148.919
C01252=1134.005,196.309,-63.475,-178.239,7.550,148.919
C01253=1134.000,196.558,-63.499,-178.235,7.552,148.919
C01254=1133.996,196.807,-63.523,-178.233,7.555,148.919
C01255=1133.990,197.056,-63.547,-178.230,7.557,148.919
C01256=1133.986,197.304,-63.572,-178.227,7.560,148.918
C01257=1133.982,197.554,-63.595,-178.224,7.563,148.918
C01258=1133.977,197.802,-63.620,-178.222,7.565,148.918
C01259=1133.972,198.051,-63.644,-178.219,7.567,148.918
C01260=1133.968,198.299,-63.668,-178.216,7.570,148.918
C01261=1133.964,198.548,-63.693,-178.213,7.572,148.917
C01262=1133.959,198.797,-63.717,-178.210,7.575,148.917
C01263=1133.954,199.046,-63.741,-178.208,7.578,148.917
C01264=1133.950,199.295,-63.765,-178.204,7.580,148.917
C01265=1133.945,199.544,-63.790,-178.202,7.583,148.917
C01266=1133.941,199.792,-63.814,-178.199,7.585,148.917
C01267=1133.934,200.166,-63.851,-178.194,7.589,148.916
C01268=1133.909,201.534,-63.985,-179.073,9.335,149.576
C01269=1133.904,201.782,-64.009,-179.069,9.338,149.575
C01270=1133.901,202.031,-64.035,-179.065,9.342,149.575
C01271=1133.896,202.280,-64.059,-179.062,9.344,149.575
C01272=1133.891,202.528,-64.085,-179.058,9.348,149.575
C01273=1133.887,202.777,-64.109,-179.055,9.351,149.575
C01274=1133.882,203.026,-64.134,-179.052,9.354,149.575
C01275=1133.878,203.274,-64.160,-179.049,9.357,149.575
C01276=1133.874,203.523,-64.184,-179.045,9.360,149.574
C01277=1133.869,203.771,-64.209,-179.043,9.363,149.575
C01278=1133.864,204.021,-64.234,-179.040,9.366,149.574
C01279=1133.859,204.270,-64.259,-179.036,9.370,149.574
C01280=1133.856,204.518,-64.284,-179.033,9.372,149.574
C01281=1133.851,204.767,-64.309,-179.030,9.375,149.574
C01282=1133.846,205.016,-64.335,-179.027,9.378,149.574
C01283=1133.841,205.264,-64.359,-179.025,9.381,149.574
C01284=1133.838,205.513,-64.384,-179.022,9.384,149.574
C01285=1133.833,205.761,-64.410,-179.019,9.386,149.574
C01286=1133.828,206.010,-64.435,-179.016,9.390,149.574
C01287=1133.824,206.258,-64.460,-179.014,9.392,149.573
C01288=1133.819,206.508,-64.485,-179.012,9.395,149.574
C01289=1133.814,206.756,-64.511,-179.009,9.397,149.573
C01290=1133.811,207.005,-64.535,-179.006,9.400,149.573
C01291=1133.806,207.253,-64.561,-179.004,9.402,149.573
C01292=1133.801,207.502,-64.586,-179.001,9.406,149.573
C01293=1133.797,207.751,-64.611,-178.999,9.408,149.573
C01294=1133.792,208.000,-64.637,-178.996,9.411,149.573
C01295=1133.788,208.248,-64.662,-178.995,9.413,149.573
C01296=1133.783,208.497,-64.687,-178.992,9.416,149.573
C01297=1133.779,208.746,-64.712,-178.990,9.418,149.573
C01298=1133.775,208.994,-64.738,-178.988,9.421,149.573
C01299=1133.770,209.243,-64.763,-178.986,9.424,149.573
C01300=1133.766,209.492,-64.788,-178.984,9.426,149.573
C01301=1133.761,209.740,-64.814,-178.982,9.428,149.574
C01302=1133.757,209.989,-64.840,-178.980,9.431,149.574
C01303=1133.752,210.238,-64.865,-178.978,9.433,149.574
C01304=1133.747,210.486,-64.890,-178.976,9.435,149.574
C01305=1133.743,210.735,-64.916,-178.974,9.438,149.574
C01306=1133.738,210.983,-64.941,-178.973,9.440,149.574
C01307=1133.734,211.232,-64.967,-178.971,9.443,149.574
C01308=1133.729,211.482,-64.992,-178.969,9.445,149.574
C01309=1133.725,211.730,-65.017,-178.968,9.448,149.574
C01310=1133.720,211.978,-65.043,-178.966,9.451,149.575
C01311=1133.716,212.227,-65.069,-178.965,9.452,149.575
C01312=1133.712,212.493,-65.095,-178.963,9.455,149.575
C01313=1133.706,212.759,-65.123,-178.962,9.458,149.575
C01314=1133.702,213.025,-65.150,-178.960,9.460,149.575
C01315=1133.697,213.290,-65.177,-178.959,9.463,149.575
C01316=1133.693,213.539,-65.202,-178.957,9.465,149.576
C01317=1133.689,213.788,-65.228,-178.956,9.468,149.576
C01318=1133.683,214.037,-65.254,-178.954,9.470,149.576
C01319=1133.679,214.285,-65.280,-178.952,9.473,149.576
C01320=1133.675,214.534,-65.306,-178.950,9.475,149.576
C01321=1133.670,214.782,-65.331,-178.949,9.478,149.576
C01322=1133.666,215.031,-65.357,-178.946,9.481,149.576
C01323=1133.661,215.280,-65.383,-178.945,9.484,149.577
C01324=1133.657,215.529,-65.408,-178.943,9.486,149.577
C01325=1133.652,215.777,-65.434,-178.941,9.490,149.577
C01326=1133.648,216.026,-65.459,-178.939,9.492,149.577
C01327=1133.644,216.275,-65.485,-178.938,9.495,149.577
C01328=1133.639,216.523,-65.511,-178.935,9.498,149.577
C01329=1133.635,216.771,-65.536,-178.933,9.501,149.578
C01330=1133.631,217.020,-65.562,-178.931,9.504,149.578
C01331=1133.626,217.269,-65.588,-178.928,9.507,149.578
C01332=1133.622,217.517,-65.613,-178.927,9.509,149.578
C01333=1133.617,217.766,-65.640,-178.924,9.512,149.578
C01334=1133.612,218.015,-65.665,-178.922,9.516,149.578
C01335=1133.608,218.264,-65.691,-178.920,9.518,149.578
C01336=1133.603,218.512,-65.716,-178.918,9.521,149.578
C01337=1133.599,218.761,-65.742,-178.915,9.524,149.578
C01338=1133.595,219.010,-65.768,-178.913,9.528,149.578
C01339=1133.591,219.258,-65.794,-178.910,9.531,149.579
C01340=1133.585,219.506,-65.820,-178.908,9.534,149.579
C01341=1133.581,219.755,-65.846,-178.905,9.537,149.579
C01342=1133.577,220.004,-65.872,-178.903,9.540,149.579
C01343=1133.573,220.253,-65.898,-178.901,9.543,149.579
C01344=1133.568,220.501,-65.923,-178.898,9.547,149.579
C01345=1133.563,220.749,-65.950,-178.896,9.550,149.579
C01346=1133.559,220.998,-65.976,-178.893,9.553,149.579
C01347=1133.555,221.247,-66.002,-178.890,9.556,149.579
C01348=1133.551,221.496,-66.027,-178.887,9.559,149.579
C01349=1133.546,221.744,-66.054,-178.884,9.563,149.579
C01350=1133.542,221.993,-66.080,-178.882,9.566,149.579
C01351=1133.537,222.241,-66.105,-178.879,9.570,149.579
C01352=1133.533,222.490,-66.131,-178.876,9.573,149.579
C01353=1133.528,222.738,-66.158,-178.873,9.575,149.579
C01354=1133.524,222.987,-66.184,-178.870,9.579,149.579
C01355=1133.520,223.236,-66.210,-178.868,9.582,149.579
C01356=1133.515,223.484,-66.237,-178.864,9.586,149.579
C01357=1133.511,223.733,-66.263,-178.861,9.589,149.579
C01358=1133.506,223.981,-66.289,-178.858,9.593,149.579
C01359=1133.501,224.230,-66.315,-178.855,9.596,149.579
C01360=1133.497,224.479,-66.341,-178.852,9.599,149.579
C01361=1133.493,224.727,-66.367,-178.849,9.603,149.579
C01362=1133.488,224.976,-66.394,-178.846,9.606,149.579
C01363=1133.484,225.224,-66.420,-178.843,9.610,149.579
C01364=1133.480,225.438,-66.442,-178.840,9.612,149.579
C01365=1133.476,225.653,-66.465,-178.837,9.615,149.579
C01366=1133.472,225.866,-66.488,-178.833,9.619,149.579
C01367=1133.469,226.081,-66.511,-178.831,9.622,149.579
C01368=1133.465,226.296,-66.534,-178.828,9.625,149.579
C01369=1133.461,226.509,-66.556,-178.825,9.628,149.579
C01370=1133.457,226.724,-66.579,-178.822,9.630,149.579
C01371=1133.453,226.938,-66.602,-178.819,9.634,149.579
C01372=1133.449,227.186,-66.629,-178.815,9.638,149.579
C01373=1133.444,227.435,-66.655,-178.812,9.641,149.578
C01374=1133.440,227.684,-66.682,-178.808,9.645,149.578
C01375=1133.436,227.933,-66.707,-178.805,9.648,149.578
C01376=1133.431,228.181,-66.734,-178.801,9.652,149.578
C01377=1133.427,228.429,-66.761,-178.797,9.655,149.578
C01378=1133.422,228.678,-66.788,-178.793,9.658,149.578
C01379=1133.418,228.927,-66.814,-178.790,9.662,149.578
C01380=1133.413,229.175,-66.841,-178.786,9.666,149.577
C01381=1133.409,229.423,-66.867,-178.782,9.669,149.577
C01382=1133.405,229.672,-66.894,-178.778,9.673,149.577
C01383=1133.400,229.921,-66.921,-178.774,9.677,149.577
C01384=1133.396,230.169,-66.947,-178.770,9.680,149.577
C01385=1133.391,230.418,-66.974,-178.766,9.684,149.577
C01386=1133.387,230.667,-67.002,-178.762,9.687,149.576
C01387=1133.383,230.915,-67.028,-178.759,9.691,149.576
C01388=1133.379,231.163,-67.055,-178.755,9.694,149.576
C01389=1133.374,231.412,-67.082,-178.751,9.697,149.576
C01390=1133.370,231.661,-67.108,-178.747,9.701,149.576
C01391=1133.365,231.909,-67.135,-178.744,9.704,149.575
C01392=1133.360,232.158,-67.162,-178.740,9.708,149.575
C01393=1133.357,232.406,-67.189,-178.737,9.710,149.575
C01394=1133.352,232.654,-67.216,-178.733,9.714,149.575
C01395=1133.347,232.903,-67.243,-178.730,9.717,149.575
C01396=1133.343,233.152,-67.270,-178.726,9.720,149.574
C01397=1133.339,233.400,-67.297,-178.723,9.723,149.574
C01398=1133.335,233.649,-67.324,-178.720,9.726,149.574
C01399=1133.330,233.897,-67.351,-178.716,9.729,149.574
C01400=1133.326,234.145,-67.378,-178.713,9.732,149.574
C01401=1133.321,234.394,-67.405,-178.710,9.735,149.574
C01402=1133.318,234.643,-67.432,-178.706,9.738,149.574
C01403=1133.313,234.891,-67.459,-178.703,9.741,149.573
C01404=1133.308,235.140,-67.486,-178.701,9.744,149.573
C01405=1133.304,235.388,-67.514,-178.698,9.746,149.573
C01406=1133.299,235.637,-67.541,-178.695,9.749,149.573
C01407=1133.295,235.885,-67.569,-178.692,9.752,149.573
C01408=1133.291,236.133,-67.595,-178.689,9.755,149.573
C01409=1133.287,236.382,-67.622,-178.686,9.757,149.573
C01410=1133.282,236.630,-67.649,-178.683,9.760,149.572
C01411=1133.277,236.879,-67.676,-178.680,9.763,149.573
C01412=1133.274,237.127,-67.705,-178.677,9.766,149.572
C01413=1133.269,237.376,-67.732,-178.674,9.769,149.572
C01414=1133.264,237.624,-67.759,-178.672,9.771,149.572
C01415=1133.260,237.873,-67.786,-178.669,9.773,149.572
C01416=1133.256,238.121,-67.814,-178.667,9.776,149.572
C01417=1133.251,238.370,-67.841,-178.664,9.779,149.572
C01418=1133.247,238.618,-67.868,-178.661,9.781,149.572
C01419=1133.243,238.866,-67.895,-178.659,9.784,149.572
C01420=1133.239,239.081,-67.919,-178.657,9.786,149.572
C01421=1133.235,239.295,-67.942,-178.655,9.788,149.572
C01422=1133.231,239.509,-67.967,-178.653,9.790,149.572
C01423=1133.228,239.723,-67.990,-178.651,9.792,149.572
C01424=1133.224,239.937,-68.014,-178.649,9.794,149.572
C01425=1133.220,240.151,-68.037,-178.647,9.796,149.572
C01426=1133.216,240.366,-68.061,-178.646,9.798,149.572
C01427=1133.213,240.579,-68.085,-178.643,9.800,149.572
C01428=1133.208,240.828,-68.112,-178.641,9.802,149.572
C01429=1133.204,241.077,-68.140,-178.639,9.805,149.572
C01430=1133.200,241.325,-68.167,-178.637,9.807,149.572
C01431=1133.195,241.573,-68.195,-178.635,9.809,149.572
C01432=1133.191,241.822,-68.222,-178.633,9.811,149.572
C01433=1133.187,242.070,-68.250,-178.631,9.814,149.572
C01434=1133.182,242.318,-68.277,-178.630,9.816,149.572
C01435=1133.179,242.567,-68.305,-178.628,9.818,149.572
C01436=1133.174,242.816,-68.332,-178.626,9.820,149.572
C01437=1133.169,243.064,-68.360,-178.625,9.822,149.572
C01438=1133.165,243.313,-68.388,-178.623,9.825,149.572
C01439=1133.160,243.561,-68.416,-178.621,9.827,149.572
C01440=1133.156,243.809,-68.443,-178.619,9.828,149.572
C01441=1133.152,244.058,-68.471,-178.618,9.831,149.572
C01442=1133.147,244.306,-68.498,-178.617,9.833,149.572
C01443=1133.143,244.554,-68.526,-178.615,9.835,149.572
C01444=1133.139,244.803,-68.553,-178.614,9.837,149.572
C01445=1133.135,245.051,-68.581,-178.612,9.839,149.573
C01446=1133.130,245.299,-68.609,-178.611,9.841,149.573
C01447=1133.125,245.549,-68.637,-178.610,9.843,149.573
C01448=1133.121,245.797,-68.664,-178.608,9.845,149.573
C01449=1133.116,246.045,-68.692,-178.607,9.847,149.573
C01450=1133.113,246.294,-68.720,-178.606,9.849,149.573
C01451=1133.108,246.542,-68.747,-178.606,9.851,149.574
C01452=1133.104,246.791,-68.775,-178.604,9.853,149.574
C01453=1133.100,247.039,-68.803,-178.603,9.855,149.574
C01454=1133.095,247.287,-68.831,-178.602,9.857,149.574
C01455=1133.091,247.536,-68.858,-178.597,9.861,149.574
C01456=1133.086,247.784,-68.886,-178.589,9.867,149.573
C01457=1133.083,248.032,-68.914,-178.582,9.873,149.573
C01458=1133.078,248.281,-68.941,-178.575,9.878,149.572
C01459=1133.073,248.529,-68.970,-178.567,9.884,149.572
C01460=1133.069,248.778,-68.998,-178.561,9.889,149.571
C01461=1133.065,249.026,-69.026,-178.553,9.894,149.570
C01462=1133.061,249.274,-69.054,-178.547,9.899,149.570
C01463=1133.056,249.522,-69.082,-178.541,9.904,149.569
C01464=1133.052,249.771,-69.110,-178.535,9.908,149.569
C01465=1133.048,250.019,-69.137,-178.530,9.911,149.568
C01466=1133.043,250.268,-69.166,-178.525,9.916,149.568
C01467=1133.039,250.516,-69.194,-178.520,9.920,149.568
C01468=1133.034,250.765,-69.223,-178.515,9.922,149.567
C01469=1133.030,251.012,-69.251,-178.511,9.926,149.567
C01470=1133.026,251.261,-69.279,-178.507,9.930,149.566
C01471=1133.022,251.510,-69.308,-178.503,9.933,149.566
C01472=1133.018,251.758,-69.336,-178.499,9.935,149.566
C01473=1133.013,252.007,-69.365,-178.496,9.938,149.566
C01474=1133.009,252.254,-69.392,-178.493,9.941,149.566
C01475=1133.004,252.503,-69.421,-178.491,9.943,149.566
C01476=1133.000,252.717,-69.446,-178.489,9.945,149.565
C01477=1132.997,252.931,-69.469,-178.487,9.947,149.565
C01478=1132.993,253.145,-69.494,-178.485,9.948,149.565
C01479=1132.990,253.359,-69.518,-178.484,9.950,149.565
C01480=1132.986,253.573,-69.544,-178.482,9.951,149.565
C01481=1132.982,253.787,-69.568,-178.482,9.952,149.565
C01482=1132.978,254.001,-69.592,-178.481,9.953,149.565
C01483=1132.975,254.215,-69.617,-178.480,9.954,149.565
C01484=1132.971,254.463,-69.645,-178.480,9.956,149.566
C01485=1132.966,254.712,-69.674,-178.480,9.956,149.566
C01486=1132.962,254.960,-69.702,-178.480,9.957,149.566
C01487=1132.958,255.208,-69.731,-178.481,9.958,149.566
C01488=1132.954,255.457,-69.759,-178.482,9.958,149.567
C01489=1132.949,255.705,-69.788,-178.483,9.958,149.567
C01490=1132.945,255.954,-69.816,-178.484,9.959,149.568
C01491=1132.940,256.202,-69.844,-178.481,9.962,149.568
C01492=1132.937,256.450,-69.873,-178.478,9.965,149.567
C01493=1132.932,256.699,-69.902,-178.476,9.968,149.568
C01494=1132.928,256.947,-69.929,-178.473,9.970,149.567
C01495=1132.923,257.196,-69.958,-178.470,9.973,149.567
C01496=1132.919,257.443,-69.987,-178.466,9.977,149.567
C01497=1132.915,257.692,-70.015,-178.463,9.979,149.567
C01498=1132.910,257.941,-70.044,-178.460,9.982,149.567
C01499=1132.906,258.188,-70.072,-178.457,9.985,149.567
C01500=1132.902,258.437,-70.101,-178.454,9.989,149.567
C01501=1132.898,258.685,-70.130,-178.451,9.991,149.567
C01502=1132.893,258.933,-70.158,-178.448,9.994,149.566
C01503=1132.889,259.182,-70.187,-178.444,9.997,149.566
C01504=1132.885,259.430,-70.215,-178.441,10.000,149.566
C01505=1132.880,259.678,-70.245,-178.438,10.004,149.566
C01506=1132.876,259.927,-70.273,-178.434,10.006,149.566
C01507=1132.872,260.175,-70.301,-178.431,10.009,149.566
C01508=1132.868,260.424,-70.331,-178.427,10.013,149.566
C01509=1132.863,260.672,-70.359,-178.424,10.015,149.565
C01510=1132.859,260.920,-70.388,-178.420,10.019,149.565
C01511=1132.855,261.169,-70.417,-178.416,10.022,149.565
C01512=1132.850,261.416,-70.446,-178.413,10.025,149.565
C01513=1132.846,261.665,-70.474,-178.409,10.028,149.565
C01514=1132.842,261.913,-70.504,-178.406,10.032,149.564
C01515=1132.837,262.162,-70.532,-178.402,10.035,149.564
C01516=1132.833,262.409,-70.561,-178.398,10.038,149.564
C01517=1132.829,262.657,-70.590,-178.394,10.041,149.564
C01518=1132.825,262.906,-70.619,-178.390,10.045,149.563
C01519=1132.821,263.155,-70.648,-178.387,10.047,149.563
C01520=1132.816,263.403,-70.678,-178.383,10.050,149.563
C01521=1132.811,263.651,-70.706,-178.379,10.053,149.563
C01522=1132.808,263.899,-70.735,-178.374,10.057,149.562
C01523=1132.804,264.147,-70.765,-178.370,10.060,149.562
C01524=1132.799,264.396,-70.793,-178.366,10.064,149.562
C01525=1132.795,264.644,-70.823,-178.364,10.066,149.562
C01526=1132.790,264.892,-70.852,-178.361,10.069,149.562
C01527=1132.786,265.140,-70.881,-178.359,10.071,149.562
C01528=1132.782,265.389,-70.910,-178.357,10.073,149.562
C01529=1132.777,265.637,-70.940,-178.354,10.075,149.561
C01530=1132.773,265.886,-70.969,-178.351,10.077,149.561
C01531=1132.770,266.134,-70.998,-178.350,10.080,149.561
C01532=1132.765,266.348,-71.023,-178.347,10.082,149.561
C01533=1132.762,266.561,-71.048,-178.345,10.084,149.561
C01534=1132.758,266.775,-71.073,-178.343,10.086,149.561
C01535=1132.755,266.990,-71.098,-178.341,10.088,149.561
C01536=1132.750,267.203,-71.124,-178.338,10.090,149.561
C01537=1132.747,267.417,-71.149,-178.336,10.092,149.561
C01538=1132.743,267.630,-71.174,-178.334,10.094,149.561
C01539=1132.740,267.845,-71.199,-178.332,10.096,149.561
C01540=1132.736,268.093,-71.229,-178.329,10.099,149.561
C01541=1132.732,268.341,-71.258,-178.327,10.101,149.560
C01542=1132.727,268.589,-71.287,-178.324,10.104,149.560
C01543=1132.723,268.837,-71.316,-178.321,10.106,149.560
C01544=1132.718,269.086,-71.346,-178.318,10.109,149.560
C01545=1132.714,269.334,-71.375,-178.316,10.111,149.560
C01546=1132.710,269.582,-71.405,-178.313,10.113,149.560
C01547=1132.706,269.830,-71.434,-178.310,10.116,149.560
C01548=1132.702,270.079,-71.464,-178.308,10.119,149.560
C01549=1132.698,270.327,-71.493,-178.305,10.121,149.560
C01550=1132.693,270.575,-71.523,-178.302,10.124,149.560
C01551=1132.688,270.824,-71.553,-178.300,10.127,149.560
C01552=1132.684,271.072,-71.582,-178.296,10.129,149.559
C01553=1132.680,271.320,-71.612,-178.293,10.132,149.559
C01554=1132.676,271.569,-71.641,-178.291,10.134,149.559
C01555=1132.672,271.817,-71.671,-178.288,10.137,149.559
C01556=1132.668,272.065,-71.700,-178.285,10.139,149.559
C01557=1132.663,272.313,-71.729,-178.282,10.142,149.559
C01558=1132.659,272.560,-71.759,-178.279,10.145,149.559
C01559=1132.655,272.809,-71.789,-178.276,10.148,149.559
C01560=1132.651,273.057,-71.818,-178.273,10.150,149.558
C01561=1132.646,273.305,-71.848,-178.270,10.153,149.558
C01562=1132.641,273.554,-71.878,-178.267,10.156,149.558
C01563=1132.638,273.801,-71.908,-178.264,10.158,149.558
C01564=1132.633,274.050,-71.937,-178.261,10.161,149.558
C01565=1132.630,274.299,-71.967,-178.258,10.164,149.558
C01566=1132.626,274.547,-71.997,-178.255,10.167,149.558
C01567=1132.621,274.795,-72.027,-178.252,10.169,149.557
C01568=1132.617,275.043,-72.057,-178.249,10.172,149.557
C01569=1132.613,275.291,-72.086,-178.246,10.174,149.557
C01570=1132.608,275.540,-72.116,-178.242,10.178,149.557
C01571=1132.605,275.787,-72.146,-178.239,10.180,149.557
C01572=1132.600,276.036,-72.176,-178.236,10.183,149.557
C01573=1132.595,276.284,-72.205,-178.233,10.186,149.556
C01574=1132.592,276.532,-72.236,-178.230,10.188,149.556
C01575=1132.587,276.780,-72.265,-178.226,10.192,149.556
C01576=1132.583,277.028,-72.296,-178.223,10.194,149.556
C01577=1132.579,277.276,-72.325,-178.220,10.197,149.556
C01578=1132.574,277.524,-72.355,-178.217,10.199,149.556
C01579=1132.570,277.772,-72.385,-178.213,10.203,149.555
C01580=1132.566,278.021,-72.415,-178.210,10.205,149.555
C01581=1132.562,278.269,-72.445,-178.206,10.208,149.555
C01582=1132.557,278.518,-72.475,-178.203,10.211,149.555
C01583=1132.554,278.765,-72.506,-178.200,10.214,149.555
C01584=1132.549,279.014,-72.535,-178.196,10.217,149.554
C01585=1132.545,279.262,-72.566,-178.193,10.220,149.554
C01586=1132.541,279.510,-72.595,-178.189,10.223,149.554
C01587=1132.537,279.757,-72.625,-178.186,10.226,149.554
C01588=1132.533,279.972,-72.652,-178.182,10.228,149.554
C01589=1132.529,280.185,-72.678,-178.179,10.231,149.553
C01590=1132.526,280.399,-72.704,-178.176,10.233,149.553
C01591=1132.522,280.613,-72.729,-178.173,10.236,149.553
C01592=1132.518,280.827,-72.756,-178.170,10.238,149.553
C01593=1132.515,281.041,-72.782,-178.167,10.240,149.552
C01594=1132.511,281.254,-72.808,-178.164,10.243,149.552
C01595=1132.508,281.468,-72.834,-178.161,10.245,149.552
C01596=1132.504,281.716,-72.865,-178.158,10.248,149.552
C01597=1132.499,281.965,-72.895,-178.154,10.250,149.552
C01598=1132.495,282.212,-72.925,-178.152,10.253,149.552
C01599=1132.490,282.460,-72.956,-178.149,10.256,149.551
C01600=1132.487,282.709,-72.986,-178.145,10.258,149.551
C01601=1132.482,282.957,-73.016,-178.142,10.261,149.551
C01602=1132.478,283.205,-73.046,-178.139,10.264,149.551
C01603=1132.474,283.453,-73.077,-178.136,10.266,149.551
C01604=1132.470,283.700,-73.107,-178.133,10.268,149.550
C01605=1132.466,283.949,-73.138,-178.130,10.271,149.550
C01606=1132.462,284.197,-73.168,-178.127,10.273,149.550
C01607=1132.457,284.445,-73.199,-178.124,10.276,149.550
C01608=1132.453,284.693,-73.229,-178.121,10.279,149.550
C01609=1132.449,284.942,-73.260,-178.118,10.281,149.550
C01610=1132.445,285.190,-73.291,-178.115,10.284,149.549
C01611=1132.441,285.437,-73.321,-178.112,10.286,149.549
C01612=1132.437,285.686,-73.352,-178.109,10.289,149.549
C01613=1132.432,285.934,-73.383,-178.105,10.291,149.549
C01614=1132.428,286.181,-73.413,-178.102,10.294,149.549
C01615=1132.423,286.430,-73.443,-178.100,10.296,149.549
C01616=1132.420,286.678,-73.474,-178.097,10.299,149.548
C01617=1132.415,286.926,-73.504,-178.094,10.301,149.548
C01618=1132.411,287.174,-73.535,-178.090,10.304,149.548
C01619=1132.407,287.423,-73.566,-178.087,10.307,149.548
C01620=1132.403,287.671,-73.596,-178.084,10.309,149.548
C01621=1132.399,287.918,-73.628,-178.081,10.312,149.547
C01622=1132.395,288.166,-73.658,-178.078,10.314,149.547
C01623=1132.391,288.414,-73.689,-178.075,10.317,149.547
C01624=1132.386,288.662,-73.720,-178.072,10.320,149.547
C01625=1132.382,288.911,-73.751,-178.069,10.322,149.547
C01626=1132.378,289.158,-73.781,-178.066,10.324,149.547
C01627=1132.374,289.406,-73.812,-178.063,10.326,149.546
C01628=1132.370,289.655,-73.843,-178.060,10.329,149.546
C01629=1132.365,289.903,-73.874,-178.057,10.332,149.546
C01630=1132.362,290.151,-73.905,-178.054,10.334,149.546
C01631=1132.357,290.399,-73.936,-178.050,10.337,149.546
C01632=1132.353,290.647,-73.967,-178.048,10.340,149.546
C01633=1132.349,290.895,-73.998,-178.044,10.342,149.545
C01634=1132.344,291.143,-74.028,-178.041,10.345,149.545
C01635=1132.341,291.391,-74.060,-178.038,10.347,149.545
C01636=1132.337,291.639,-74.091,-178.035,10.350,149.545
C01637=1132.332,291.887,-74.121,-178.032,10.353,149.545
C01638=1132.328,292.136,-74.152,-178.029,10.354,149.544
C01639=1132.324,292.383,-74.184,-178.026,10.357,149.544
C01640=1132.320,292.631,-74.214,-178.023,10.360,149.544
C01641=1132.316,292.879,-74.245,-178.020,10.362,149.544
C01642=1132.312,293.127,-74.277,-178.017,10.365,149.544
C01643=1132.307,293.375,-74.308,-178.014,10.368,149.544
C01644=1132.304,293.589,-74.335,-178.011,10.369,149.543
C01645=1132.301,293.803,-74.362,-178.008,10.372,149.543
C01646=1132.297,294.016,-74.388,-178.006,10.374,149.543
C01647=1132.293,294.230,-74.415,-178.003,10.377,149.543
C01648=1132.290,294.444,-74.442,-178.000,10.378,149.543
C01649=1132.286,294.657,-74.469,-177.998,10.380,149.543
C01650=1132.283,294.870,-74.496,-177.995,10.383,149.543
C01651=1132.279,295.084,-74.523,-177.992,10.385,149.542
C01652=1132.275,295.332,-74.554,-177.989,10.387,149.542
C01653=1132.271,295.580,-74.585,-177.986,10.390,149.542
C01654=1132.267,295.828,-74.616,-177.983,10.393,149.542
C01655=1132.263,296.076,-74.648,-177.980,10.395,149.542
C01656=1132.259,296.324,-74.679,-177.977,10.398,149.541
C01657=1132.254,296.572,-74.710,-177.973,10.400,149.541
C01658=1132.250,296.820,-74.742,-177.971,10.403,149.541
C01659=1132.246,297.068,-74.773,-177.968,10.405,149.541
C01660=1132.242,297.316,-74.804,-177.965,10.407,149.541
C01661=1132.238,297.564,-74.836,-177.962,10.410,149.540
C01662=1132.234,297.812,-74.867,-177.959,10.413,149.540
C01663=1132.229,298.060,-74.898,-177.955,10.415,149.540
C01664=1132.226,298.308,-74.930,-177.952,10.418,149.540
C01665=1132.220,298.556,-74.961,-177.949,10.420,149.540
C01666=1132.217,298.804,-74.993,-177.946,10.423,149.540
C01667=1132.213,299.052,-75.025,-177.943,10.425,149.539
C01668=1132.208,299.300,-75.056,-177.940,10.428,149.539
C01669=1132.205,299.548,-75.088,-177.936,10.431,149.539
C01670=1132.200,299.795,-75.119,-177.934,10.433,149.539
C01671=1132.196,300.044,-75.150,-177.930,10.436,149.539
C01672=1132.193,300.292,-75.182,-177.927,10.439,149.539
C01673=1132.188,300.540,-75.214,-177.925,10.440,149.538
C01674=1132.184,300.788,-75.246,-177.922,10.443,149.538
C01675=1132.180,301.035,-75.278,-177.918,10.445,149.538
C01676=1132.176,301.284,-75.309,-177.915,10.448,149.538
C01677=1132.172,301.532,-75.341,-177.912,10.451,149.538
C01678=1132.168,301.779,-75.372,-177.909,10.453,149.537
C01679=1132.163,302.028,-75.405,-177.906,10.456,149.537
C01680=1132.159,302.276,-75.436,-177.903,10.459,149.537
C01681=1132.155,302.524,-75.467,-177.900,10.461,149.537
C01682=1132.151,302.772,-75.499,-177.897,10.464,149.537
C01683=1132.147,303.019,-75.530,-177.893,10.466,149.537
C01684=1132.142,303.267,-75.563,-177.890,10.469,149.536
C01685=1132.139,303.515,-75.595,-177.887,10.471,149.536
C01686=1132.134,303.763,-75.626,-177.884,10.474,149.536
C01687=1132.130,304.011,-75.659,-177.881,10.477,149.536
C01688=1132.126,304.259,-75.691,-177.878,10.478,149.536
C01689=1132.122,304.506,-75.722,-177.875,10.481,149.535
C01690=1132.118,304.754,-75.754,-177.872,10.484,149.535
C01691=1132.114,305.003,-75.786,-177.869,10.486,149.535
C01692=1132.110,305.251,-75.818,-177.865,10.489,149.535
C01693=1132.106,305.498,-75.850,-177.863,10.491,149.535
C01694=1132.101,305.747,-75.882,-177.859,10.494,149.535
C01695=1132.098,305.995,-75.914,-177.856,10.496,149.534
C01696=1132.093,306.242,-75.945,-177.853,10.499,149.534
C01697=1132.089,306.490,-75.978,-177.850,10.502,149.534
C01698=1132.085,306.738,-76.010,-177.847,10.504,149.534
C01699=1132.081,306.987,-76.042,-177.843,10.507,149.534
C01700=1132.078,307.200,-76.070,-177.841,10.509,149.533
C01701=1132.074,307.413,-76.097,-177.838,10.512,149.533
C01702=1132.070,307.626,-76.125,-177.835,10.513,149.533
C01703=1132.067,307.840,-76.152,-177.833,10.515,149.533
C01704=1132.063,308.053,-76.180,-177.830,10.518,149.533
C01705=1132.060,308.266,-76.208,-177.828,10.520,149.533
C01706=1132.056,308.480,-76.236,-177.825,10.522,149.533
C01707=1132.053,308.693,-76.263,-177.822,10.524,149.532
C01708=1132.048,308.941,-76.296,-177.819,10.527,149.532
C01709=1132.045,309.189,-76.328,-177.816,10.529,149.532
C01710=1132.040,309.438,-76.360,-177.813,10.532,149.532
C01711=1132.036,309.685,-76.392,-177.809,10.534,149.532
C01712=1132.032,309.933,-76.425,-177.806,10.537,149.532
C01713=1132.028,310.181,-76.457,-177.803,10.540,149.531
C01714=1132.024,310.429,-76.490,-177.800,10.542,149.531
C01715=1132.020,310.677,-76.522,-177.797,10.544,149.531
C01716=1132.016,310.925,-76.554,-177.794,10.546,149.531
C01717=1132.012,311.172,-76.586,-177.791,10.549,149.531
C01718=1132.007,311.420,-76.619,-177.788,10.552,149.530
C01719=1132.004,311.668,-76.651,-177.785,10.554,149.530
C01720=1131.999,311.916,-76.684,-177.782,10.557,149.530
C01721=1131.996,312.164,-76.716,-177.778,10.559,149.530
C01722=1131.992,312.412,-76.749,-177.775,10.562,149.530
C01723=1131.988,312.660,-76.781,-177.772,10.565,149.529
C01724=1131.983,312.907,-76.813,-177.769,10.567,149.529
C01725=1131.979,313.155,-76.846,-177.766,10.570,149.529
C01726=1131.975,313.403,-76.878,-177.762,10.572,149.529
C01727=1131.971,313.651,-76.911,-177.760,10.575,149.529
C01728=1131.967,313.899,-76.943,-177.756,10.577,149.528
C01729=1131.963,314.147,-76.976,-177.753,10.580,149.528
C01730=1131.959,314.394,-77.009,-177.750,10.583,149.528
C01731=1131.955,314.642,-77.041,-177.747,10.585,149.528
C01732=1131.951,314.890,-77.074,-177.744,10.588,149.528
C01733=1131.947,315.138,-77.106,-177.741,10.589,149.527
C01734=1131.943,315.386,-77.139,-177.738,10.592,149.527
C01735=1131.938,315.633,-77.172,-177.735,10.595,149.527
C01736=1131.934,315.881,-77.204,-177.731,10.597,149.527
C01737=1131.931,316.129,-77.237,-177.728,10.600,149.527
C01738=1131.926,316.377,-77.269,-177.725,10.602,149.527
C01739=1131.922,316.625,-77.302,-177.722,10.605,149.526
C01740=1131.919,316.872,-77.335,-177.719,10.608,149.526
C01741=1131.914,317.120,-77.368,-177.716,10.610,149.526
C01742=1131.910,317.368,-77.400,-177.712,10.612,149.526
C01743=1131.906,317.616,-77.434,-177.709,10.615,149.526
C01744=1131.903,317.863,-77.466,-177.706,10.618,149.525
C01745=1131.898,318.112,-77.499,-177.703,10.620,149.525
C01746=1131.894,318.359,-77.532,-177.700,10.623,149.525
C01747=1131.890,318.607,-77.565,-177.696,10.625,149.525
C01748=1131.886,318.855,-77.598,-177.693,10.628,149.525
C01749=1131.882,319.102,-77.631,-177.690,10.631,149.525
C01750=1131.878,319.351,-77.663,-177.687,10.633,149.524
C01751=1131.874,319.598,-77.696,-177.684,10.636,149.524
C01752=1131.870,319.846,-77.729,-177.681,10.638,149.524
C01753=1131.866,320.094,-77.762,-177.677,10.641,149.524
C01754=1131.862,320.341,-77.795,-177.675,10.643,149.524
C01755=1131.858,320.589,-77.828,-177.672,10.645,149.523
C01756=1131.855,320.803,-77.857,-177.669,10.648,149.523
C01757=1131.851,321.016,-77.886,-177.666,10.649,149.523
C01758=1131.847,321.230,-77.914,-177.663,10.652,149.523
C01759=1131.844,321.442,-77.942,-177.660,10.654,149.523
C01760=1131.841,321.656,-77.970,-177.658,10.656,149.523
C01761=1131.838,321.869,-78.000,-177.655,10.658,149.522
C01762=1131.834,322.083,-78.028,-177.652,10.660,149.522
C01763=1131.830,322.296,-78.057,-177.650,10.663,149.522
C01764=1131.826,322.543,-78.090,-177.646,10.666,149.522
C01765=1131.822,322.791,-78.123,-177.643,10.668,149.522
C01766=1131.818,323.039,-78.156,-177.640,10.671,149.522
C01767=1131.814,323.287,-78.189,-177.637,10.672,149.521
C01768=1131.811,323.535,-78.222,-177.634,10.675,149.521
C01769=1131.807,323.782,-78.255,-177.631,10.678,149.521
C01770=1131.803,324.030,-78.288,-177.628,10.680,149.521
C01771=1131.799,324.278,-78.322,-177.624,10.683,149.520
C01772=1131.794,324.526,-78.355,-177.621,10.685,149.520
C01773=1131.790,324.773,-78.388,-177.618,10.688,149.520
C01774=1131.787,325.020,-78.422,-177.615,10.690,149.520
C01775=1131.782,325.268,-78.455,-177.611,10.693,149.520
C01776=1131.779,325.517,-78.489,-177.609,10.695,149.520
C01777=1131.774,325.765,-78.522,-177.605,10.698,149.519
C01778=1131.770,326.012,-78.555,-177.602,10.700,149.519
C01779=1131.766,326.259,-78.589,-177.599,10.703,149.519
C01780=1131.762,326.507,-78.622,-177.596,10.706,149.519
C01781=1131.758,326.755,-78.656,-177.592,10.708,149.519
C01782=1131.754,327.003,-78.689,-177.589,10.711,149.519
C01783=1131.750,327.250,-78.723,-177.586,10.713,149.518
C01784=1131.746,327.498,-78.756,-177.583,10.716,149.518
C01785=1131.742,327.746,-78.789,-177.579,10.718,149.518
C01786=1131.738,327.993,-78.823,-177.577,10.721,149.518
C01787=1131.735,328.241,-78.857,-177.573,10.723,149.517
C01788=1131.730,328.490,-78.890,-177.570,10.726,149.517
C01789=1131.726,328.737,-78.924,-177.567,10.729,149.517
C01790=1131.722,328.984,-78.957,-177.564,10.731,149.517
C01791=1131.719,329.232,-78.992,-177.561,10.733,149.517
C01792=1131.714,329.480,-79.025,-177.558,10.735,149.516
C01793=1131.710,329.728,-79.058,-177.555,10.738,149.516
C01794=1131.706,329.975,-79.092,-177.551,10.740,149.516
C01795=1131.702,330.224,-79.126,-177.548,10.743,149.516
C01796=1131.698,330.471,-79.160,-177.545,10.746,149.516
C01797=1131.694,330.718,-79.193,-177.542,10.748,149.516
C01798=1131.690,330.966,-79.228,-177.538,10.750,149.515
C01799=1131.686,331.214,-79.261,-177.535,10.753,149.515
C01800=1131.682,331.461,-79.295,-177.532,10.756,149.515
C01801=1131.678,331.709,-79.328,-177.529,10.758,149.515
C01802=1131.674,331.956,-79.363,-177.526,10.761,149.515
C01803=1131.670,332.205,-79.396,-177.522,10.763,149.514
C01804=1131.666,332.452,-79.430,-177.519,10.766,149.514
C01805=1131.662,332.699,-79.464,-177.516,10.768,149.514
C01806=1131.658,332.948,-79.498,-177.513,10.771,149.514
C01807=1131.654,333.195,-79.532,-177.509,10.773,149.513
C01808=1131.650,333.442,-79.566,-177.506,10.776,149.513
C01809=1131.646,333.691,-79.600,-177.503,10.778,149.513
C01810=1131.642,333.938,-79.634,-177.500,10.781,149.513
C01811=1131.639,334.185,-79.668,-177.497,10.783,149.513
C01812=1131.635,334.399,-79.697,-177.494,10.785,149.513
C01813=1131.631,334.612,-79.726,-177.491,10.788,149.512
C01814=1131.628,334.825,-79.755,-177.489,10.790,149.512
C01815=1131.625,335.038,-79.784,-177.486,10.791,149.512
C01816=1131.621,335.251,-79.813,-177.483,10.794,149.512
C01817=1131.618,335.464,-79.844,-177.480,10.796,149.512
C01818=1131.615,335.677,-79.873,-177.477,10.799,149.512
C01819=1131.612,335.891,-79.902,-177.475,10.800,149.511
C01820=1131.607,336.138,-79.936,-177.471,10.803,149.511
C01821=1131.603,336.385,-79.970,-177.468,10.806,149.511
C01822=1131.599,336.634,-80.004,-177.465,10.808,149.511
